# B&R Automation Studio project 2x1HWDemo (part 2)

### GlobalTypes.typ
```iecst
(*Main System Interface Types*)

TYPE
	MainIfTyp : 	STRUCT
		Cmd : MainIfCmdTyp;
		Par : MainIfParTyp;
		Cfg : MainIfCfgTyp;
		Status : MainIfStatusTyp;
	END_STRUCT;
	MainIfCmdTyp : 	STRUCT
		Power : BOOL;
		Start : BOOL;
		Stop : BOOL;
		Reset : BOOL;
	END_STRUCT;
	MainIfParTyp : 	STRUCT
		Tmp : USINT;
	END_STRUCT;
	MainIfCfgTyp : 	STRUCT
		ShuttleCount : USINT;
	END_STRUCT;
	MainIfStatusTyp : 	STRUCT
		PowerOn : BOOL;
		Running : BOOL;
		Error : BOOL;
	END_STRUCT;
END_TYPE

(*Process Info Interface*)

TYPE
	ProcessInfoIfTyp : 	STRUCT
		Cmd : ProcessInfoIfCmdTyp;
		Par : ProcessInfoIfParTyp;
		Sts : ProcessInfoIfStsTyp;
	END_STRUCT;
	ProcessInfoIfCmdTyp : 	STRUCT
		Enable : BOOL;
		ResetData : BOOL;
	END_STRUCT;
	ProcessInfoIfParTyp : 	STRUCT
		CurrentProductCount : UDINT;
	END_STRUCT;
	ProcessInfoIfStsTyp : 	STRUCT
		Enabled : BOOL;
		CurrentPPM : REAL;
		CurrentPPH : REAL;
		CurrentBlistersPerMinute : REAL;
		CurrentLayersPerMinute : REAL;
	END_STRUCT;
END_TYPE

(*6D Controller Interface Types*)

TYPE
	Acp6DCmdType : 	STRUCT
		Power : BOOL;
		ErrorReset : BOOL;
		GetErrorInfo : BOOL;
	END_STRUCT;
	Acp6DCtrlType : 	STRUCT
		Cmd : Acp6DCmdType;
		Status : Acp6DStatusType;
		Par : Acp6DParType;
	END_STRUCT;
	Acp6DParType : 	STRUCT
		Mode : McAcp6DMoveModeEnum;
		PathType : McAcp6DInPlaneMovePathEnum;
		Acceleration : REAL;
		EndVelocity : REAL;
		Velocity : REAL;
		ShuttleID : USINT;
		SegmentID : USINT;
		PositionX : REAL;
		PositionY : REAL;
	END_STRUCT;
	Acp6DStatusType : 	STRUCT
		Error : BOOL;
		ErrorID : DINT;
		Ready : BOOL;
		PowerOn : BOOL;
		ReadyToPowerOn : BOOL;
		ErrorCodes : ARRAY[0..8]OF DINT;
	END_STRUCT;
	Acp6DShuttleInfoType : 	STRUCT
		State : Acp6DShuttleStateInfoTyp;
		Force : Acp6DShuttleForceInfoTyp;
		Position : Acp6DShuttlePosInfoTyp;
	END_STRUCT;
	Acp6DShuttleStateInfoTyp : 	STRUCT
		Valid : BOOL;
		Value : McAcp6DShuttleStateEnum;
	END_STRUCT;
	Acp6DShuttlePosInfoTyp : 	STRUCT
		Valid : BOOL;
		Value : McAcp6DShPositionInfoType;
	END_STRUCT;
	Acp6DShuttleForceInfoTyp : 	STRUCT
		Valid : BOOL;
		Value : McAcp6DShForceInfoType;
	END_STRUCT;
END_TYPE

(*Shuttle Interface Types*)

TYPE
	gShuttleIfCmdTyp : 	STRUCT  (*Commands for controlling a shuttle*)
		Enable : BOOL; (*Command for enabling the control of a shuttle in the process*)
		Recover : BOOL; (*Command for a shuttle to start recovery*)
		NextStep : BOOL; (*Command for a shuttle to start the next step in the process*)
		ResetProductInfo : BOOL; (*Command to reset all the product info on a shuttle*)
		Stop : BOOL; (*Command to stop the process for a shuttle*)
	END_STRUCT;
	gShuttleIfCfgMacrosTyp : 	STRUCT  (*Structure of the macro IDs used for operation*)
		RobotProcessMacro : gShuttleIfMacroEnum; (*Macro ID used for sending a shuttle from the load station to the print station*)
	END_STRUCT;
	gShuttleIfParTyp : 	STRUCT  (*Parameters for the shuttle's operation*)
		NumLayers : USINT; (*Number of layers for this defined recipe*)
		MacroIDs : gShuttleIfCfgMacrosTyp; (*Macro's used for routing shuttles*)
	END_STRUCT;
	gShuttleIfConfigTyp : 	STRUCT  (*Configuration values for a shuttle*)
		ShuttleId : USINT; (*ShuttleID of this shuttle*)
	END_STRUCT;
	gShuttleIfMacroEnum :
		( (*Macro IDs that are used to denote which macro means what*)
		MACRO_ROBOT_PROCESS := 128, (*Macro ID used for sending a shuttle from the load station to the print station*)
		MACRO_RECOVERY_GROUP0 (*Macro ID used for recovering the group 0 shuttles*)
		);
	gShuttleIfDestEnum :
		( (*Destinations for a shuttle to move to*)
		DEST_LOAD, (*Destination Load station*)
		DEST_PRINT, (*Destination Printing station*)
		DEST_DOSE1, (*Destination Dose 1 station*)
		DEST_DOSE2, (*Destination Dose 2 station*)
		DEST_TAMP, (*Destination Tamping station*)
		DEST_UNLOAD (*Destination unload*)
		);
	ShStateEnum :
		(
		SH_OFF, (*Shuttle is in the off/idle state*)
		SH_INIT, (*Shuttle is in the initilization state*)
		SH_STARTUP, (*Shuttle is in the startup state*)
		SH_IDLE, (*Shuttle is in the idle state after having been recovered*)
		SH_MOVE_TO_ROBOT,
		SH_ROBOT,
		SH_OFFLOAD, (*Shuttle is currently being offloaded*)
		SH_ERROR := 65535 (*Shuttle is in the error state*)
		);
	gShuttleIfStatusTyp : 	STRUCT  (*Status information for the shuttle*)
		CurrentDestination : gShuttleIfDestEnum; (*Destination the shuttle is currently moving towards*)
		ShuttleInfo : Acp6DShuttleInfoType; (*CurrentStatus Information about the shuttle*)
		Error : BOOL; (*Shuttle is currently in an error state*)
		ErrorState : ShStateEnum; (*State the shuttle errored at*)
		Recovered : BOOL; (*Shuttle has been recovered*)
		CyclicPositionX : REAL;
	END_STRUCT;
	gShuttleIfTyp : 	STRUCT  (*Interface for controlling a shuttle*)
		Cmd : gShuttleIfCmdTyp; (*Commands to issue to a shuttle*)
		Par : gShuttleIfParTyp; (*Parameters for the process for this shuttle*)
		Cfg : gShuttleIfConfigTyp; (*Configuration values for this shuttle*)
		Status : gShuttleIfStatusTyp; (*Status information related to this shuttle*)
	END_STRUCT;
END_TYPE

(*Robot Interface Types*)

TYPE
	RobotIfTyp : 	STRUCT
		Cmds : RobotIfCmdsTyp;
		Pars : RobotIfParsTyp;
		Status : RobotIfStatusTyp;
	END_STRUCT;
	RobotIfCmdsTyp : 	STRUCT
		Admin : RobotIfAdminCmdsTyp;
		Process : RobotIfProcessCmdsTyp;
	END_STRUCT;
	RobotIfAdminCmdsTyp : 	STRUCT
		Power : BOOL;
		Home : BOOL;
		Reset : BOOL;
	END_STRUCT;
	RobotIfProcessCmdsTyp : 	STRUCT
		MoveToSync : BOOL;
		Sync : BOOL;
		UnSync : BOOL;
		Run : BOOL;
	END_STRUCT;
	RobotIfParsTyp : 	STRUCT
		SyncPosition : McPosType;
		SyncFrame : STRING[80];
		SyncFrameIdent : UDINT;
		MoveToSyncVel : LREAL;
		MoveToSyncAccel : LREAL;
		MoveToSyncDecel : LREAL;
		ShuttleIdx : USINT;
	END_STRUCT;
	RobotIfStatusTyp : 	STRUCT
		Synced : BOOL;
		Homed : BOOL;
		Powered : BOOL;
		AtSync : BOOL;
	END_STRUCT;
	SceneViewerTyp : 	STRUCT
		Cmds : SceneViewerCmdsTyp;
		Pars : SceneViewerParsTyp;
	END_STRUCT;
	SceneViewerCmdsTyp : 	STRUCT
		Record : BOOL;
		Clear : BOOL;
	END_STRUCT;
	SceneViewerParsTyp : 	STRUCT
		LineColor : SceneViewerColorTyp;
	END_STRUCT;
	SceneViewerColorTyp : 	STRUCT
		Red : REAL;
		Green : REAL;
		Blue : REAL;
	END_STRUCT;
END_TYPE

(*Sync Interface Types*)

TYPE
	SyncSecIfTyp : 	STRUCT
		Cmds : SyncSecCmdsIfTyp;
		Pars : USINT;
		Status : SyncSecIfStatusTyp;
	END_STRUCT;
	SyncSecCmdsIfTyp : 	STRUCT
		Admin : SyncSecIfAdminCmdsTyp;
		Proc : SyncSecIfProcCmdsTyp;
	END_STRUCT;
	SyncSecIfAdminCmdsTyp : 	STRUCT
		New_Member : USINT;
	END_STRUCT;
	SyncSecIfProcCmdsTyp : 	STRUCT
		Start : BOOL;
		Stop : BOOL;
		ReleaseSync : BOOL;
		ReleaseUnSync : BOOL;
	END_STRUCT;
	SyncSecIfStatusTyp : 	STRUCT
		Running : BOOL;
		SyncReady : BOOL;
		UnsyncReady : BOOL;
		Error : BOOL;
		AxisToSync : McAxisType;
	END_STRUCT;
	SyncSecStatusEnum :
		(
		SYNC_OFF,
		SYNC_INIT,
		SYNC_RUNNING,
		SYNC_STOPPING,
		SYNC_ERROR
		);
END_TYPE

(*Recovery Interface Type*)

TYPE
	Acp6DRecoveryIfTyp : 	STRUCT
		Cmd : Acp6DRecoveryCmdTyp;
		Par : Acp6DRecoveryParTyp;
		Sts : Acp6DRecoveryStsTyp;
	END_STRUCT;
	Acp6DRecoveryCmdTyp : 	STRUCT
		Recover : BOOL;
		Reset : BOOL;
	END_STRUCT;
	Acp6DRecoveryParTyp : 	STRUCT
		AutoDrivePositions : ARRAY[0..MAX_SHUTTLE_COUNT_ARRAY]OF Acp6DAutoDrivePosTyp;
		Vel : REAL;
		Accel : REAL;
	END_STRUCT;
	Acp6DRecoveryStsTyp : 	STRUCT
		Recovering : BOOL;
		ReadyToStartProc : BOOL;
		Done : BOOL;
		ShuttlesRecovered : BOOL;
		Error : BOOL;
	END_STRUCT;
	Acp6DAutoDrivePosTyp : 	STRUCT
		ShIdx : USINT;
		GroupNum : USINT; (*Group ID used for recovery. Lower group, lower priority*)
		X : REAL;
		Y : REAL;
	END_STRUCT;
END_TYPE

(***********************Station Types*)
(*Load Station Types*)

TYPE
	LoadStationIfTyp : 	STRUCT
		Cmd : LoadStationCmdTyp; (*Commands to the station*)
		Par : LoadStationParTyp; (*Paramters for the station's operation*)
		Cfg : LoadStationCfgTyp; (*Configuration values for the station*)
		Status : LoadStationStatusTyp; (*Status of the station*)
	END_STRUCT;
	LoadStationCmdTyp : 	STRUCT
		Enable : BOOL; (*Enables the process station*)
		Process : BOOL; (*Start a process for the station with the defined shuttle index*)
		Reset : BOOL; (*Resets the process from an any state*)
	END_STRUCT;
	LoadStationParTyp : 	STRUCT
		ShuttleIdx : USINT; (*Index in the gShuttle array for the shuttle in question*)
		WaitTime : TIME; (*Amount of time to wait for the load process*)
	END_STRUCT;
	LoadStationCfgTyp : 	STRUCT
		StationPos : StationPositionTyp; (*Station's center world position*)
	END_STRUCT;
	LoadStationStatusTyp : 	STRUCT
		Enabled : BOOL; (*Signal denoting the station is enabled and in an operational state*)
		Processing : BOOL; (*Signal denoting the station is currently operating on a shuttle*)
		Done : BOOL; (*Signal denoting the current operation has completed*)
		ReadyForNewShuttle : BOOL; (*Signal denoting the station is ready for a new shuttle*)
		Error : BOOL; (*Signal denoting the station has an error present*)
	END_STRUCT;
	StationPositionTyp : 	STRUCT
		X : REAL; (*Station's Global X position*)
		Y : REAL; (*Station's Global Y position*)
	END_STRUCT;
END_TYPE

(*Pick Place Types*)

TYPE
	posTyp : 	STRUCT
		X : LREAL;
		Y : LREAL;
		Z : LREAL;
	END_STRUCT;
	RobotPickPlaceParsTyp : 	STRUCT
		PickTune : pickTuneTyp;
		PlaceTune : pickTuneTyp;
		ReadyPos : posTyp;
		ProductSpeed : robotSpeedTyp;
		EmptySpeed : robotSpeedTyp;
	END_STRUCT;
	pickTuneTyp : 	STRUCT
		ApproachHeight : LREAL;
		DepartHeight : LREAL;
		XTune : LREAL;
		YTune : LREAL;
		ZTune : LREAL;
		Radius : LREAL;
		DwellTime : REAL;
	END_STRUCT;
	robotSpeedTyp : 	STRUCT
		Vel : REAL;
		Accel : REAL;
		Decel : REAL;
	END_STRUCT;
	RobotPickPlaceStatusTyp : 	STRUCT
		ProductOK : BOOL;
		ProductPresent : BOOL;
		AtSync : BOOL;
	END_STRUCT;
	RobotPickPlaceCfgTyp : 	STRUCT
		PlaceLoc : posTyp;
		PickLoc : posTyp;
		SyncLoc : posTyp;
	END_STRUCT;
	RobotPickPlaceTyp : 	STRUCT
		Run : BOOL;
		Sync : BOOL;
		Config : RobotPickPlaceCfgTyp;
		Pars : RobotPickPlaceParsTyp;
		Status : RobotPickPlaceStatusTyp;
	END_STRUCT;
END_TYPE
```

### Package Logical/Source/ShuttleCtrl - Package that contains code for controlling individual shuttles

### Program Logical/Source/ShuttleCtrl/ShCtrl (IEC)

#### Types.typ
```iecst
TYPE
	ShFbsTyp : 	STRUCT
		ShRunMacroFb : MC_BR_MacroRun_Acp6D; (*Execute a macro on the current shuttle*)
		ReadCyclicPos : MC_BR_ReadCyclicChAxis_Acp6D;
	END_STRUCT;
END_TYPE
```

#### Variables.var
```iecst
VAR
	i : USINT; (*Loop index*)
	shState : ARRAY[0..MAX_SHUTTLE_COUNT_ARRAY] OF ShStateEnum;
	shFbs : ARRAY[0..MAX_SHUTTLE_COUNT_ARRAY] OF ShFbsTyp;
	pDebugIf : REFERENCE TO gShuttleIfTyp;
	pDebugFbs : REFERENCE TO ShFbsTyp;
	pDebugState : REFERENCE TO ShStateEnum;
	debugIdx : USINT;
END_VAR
```

#### Cyclic.st
```iecst
PROGRAM _CYCLIC
	FOR i:= 0 TO gMainIf.Cfg.ShuttleCount - 1 DO

		CASE shState[i] OF
			SH_OFF:  //******************************************************************************** Shuttle is in the off/idle state
				IF gShuttleIf[i].Cmd.Enable THEN
					shState[i] := SH_INIT;
				ELSE

				END_IF
			SH_INIT:  //******************************************************************************** Shuttle is in the initilization state
				//In this state we could make any checks on the current shuttle process perhaps in order to aide in recovery?
				shFbs[i].ReadCyclicPos.Controller := ADR(gMcAcp6DController);
				shFbs[i].ReadCyclicPos.ChannelID := i + 1;
				shFbs[i].ReadCyclicPos.AxisID := 1;
				shFbs[i].ReadCyclicPos.Enable := TRUE;

				shState[i] := SH_STARTUP;
			SH_STARTUP:  //******************************************************************************** Shuttle is in the startup state
				//In this state maybe we have triggered recovery and we're waiting for the autodrive to complete
				IF shFbs[i].ReadCyclicPos.Valid THEN
					shState[i] := SH_IDLE;
				END_IF
			SH_IDLE:  //******************************************************************************** Shuttle is in the idle state
				IF gShuttleIf[i].Cmd.NextStep THEN
					gShuttleIf[i].Cmd.NextStep := FALSE;
					//Evaluate the current step to determine what the next step should be
					shFbs[i].ShRunMacroFb.Controller := ADR(gMcAcp6DController);
					shFbs[i].ShRunMacroFb.ShuttleID := gShuttleIf[i].Cfg.ShuttleId;
					shFbs[i].ShRunMacroFb.MacroID := UDINT_TO_USINT(gShuttleIf[i].Par.MacroIDs.RobotProcessMacro);
					shFbs[i].ShRunMacroFb.Execute := TRUE;
					gShuttleIf[i].Status.CurrentDestination := DEST_LOAD;
					LogDebug(gAuditTrail,i,"Sent to Robot");

					shState[i] := SH_MOVE_TO_ROBOT;
				END_IF
			SH_MOVE_TO_ROBOT:  //******************************************************************************** Shuttle is moving to the load position
				IF shFbs[i].ShRunMacroFb.Error THEN
					gShuttleIf[i].Status.Error := TRUE;
					gShuttleIf[i].Status.ErrorState := shState[i];
					shState[i] := SH_ERROR;
				ELSIF shFbs[i].ShRunMacroFb.Acknowledge THEN //Check to see if the shuttle is ready to sync with the robot
					gLoadStationIf.Par.ShuttleIdx := i;
					gLoadStationIf.Cmd.Process := TRUE;

					LogDebug(gAuditTrail,i,"Arrived at Robot");

					shFbs[i].ShRunMacroFb.Execute := FALSE;
					shState[i] := SH_ROBOT;
				END_IF
			SH_ROBOT:  //******************************************************************************** Shuttle is currently being loaded
				//Station has control on the shuttle during this section
				IF gShuttleIf[i].Cmd.NextStep THEN
					gLoadStationIf.Cmd.Process := FALSE; //Respond to the Load station we're done

					gShuttleIf[i].Cmd.NextStep := FALSE;
					gShuttleIf[i].Status.CurrentDestination := DEST_PRINT;

					LogDebug(gAuditTrail,i,"Finished with Robot");

					shState[i] := SH_MOVE_TO_ROBOT;
				END_IF

			SH_ERROR: //******************************************************************************** Shuttle is in the error state

		END_CASE;
		shFbs[i].ShRunMacroFb();

		IF gShuttleIf[i].Cmd.ResetProductInfo THEN
			gShuttleIf[i].Status.Error := FALSE;
			gShuttleIf[i].Status.ErrorState := 0;
			gShuttleIf[i].Cmd.ResetProductInfo := FALSE;
		END_IF
	END_FOR;
	pDebugIf ACCESS ADR(gShuttleIf[debugIdx]);
	pDebugState ACCESS ADR(shState[debugIdx]);
	pDebugFbs ACCESS ADR(shFbs[debugIdx]);

END_PROGRAM
```

#### Init.st
```iecst
PROGRAM _INIT
	FOR i:=0 TO MAX_SHUTTLE_COUNT-1 DO
		gShuttleIf[i].Par.MacroIDs.RobotProcessMacro := MACRO_ROBOT_PROCESS;

	END_FOR;
END_PROGRAM
```

### Program Logical/Source/ShuttleCtrl/Recovery (IEC)

#### Init.st
```iecst
PROGRAM _INIT
	g6DRecoveryIf.Par.Vel := 1;
	g6DRecoveryIf.Par.Accel := 10;

	//************************************************************************* Shuttle 1
	g6DRecoveryIf.Par.AutoDrivePositions[0].ShIdx := 0;
	g6DRecoveryIf.Par.AutoDrivePositions[0].GroupNum := 0;
	g6DRecoveryIf.Par.AutoDrivePositions[0].X := 0.12;
	g6DRecoveryIf.Par.AutoDrivePositions[0].Y := 0.12;
	//************************************************************************* Shuttle 2
	g6DRecoveryIf.Par.AutoDrivePositions[1].ShIdx := 1;
	g6DRecoveryIf.Par.AutoDrivePositions[1].GroupNum := 0;
	g6DRecoveryIf.Par.AutoDrivePositions[1].X := 0.36;
	g6DRecoveryIf.Par.AutoDrivePositions[1].Y := 0.12;

END_PROGRAM
```

### Program Logical/Source/ShuttleCtrl/KalmanTesting (IEC)

#### Types.typ
```iecst
TYPE
	WeighTyp : 	STRUCT
		TareWeight : REAL;
		ExpectedWeight : REAL;
		Error : REAL;
		CalculatedExpectedForce : REAL;
		CalcWeight : REAL;
		TriggerThreshold : REAL;
	END_STRUCT;
END_TYPE
```

#### Variables.var
```iecst
VAR
	readCyclicForceFb : MC_BR_ReadCyclicChAxis_Acp6D;
	weighKalman : WFPredictiveFilter;
	WeighFb : MC_BR_GetPayload_Acp6D;
	OutputCovertedToWeight : ARRAY[0..1] OF LREAL;
	filterTest : BOOL;
	WeightTest : BOOL;
	enableFilters : BOOL;
	state : INT;
	KalmanFb : ARRAY[0..1] OF MTFilterKalman;
	ExpectedWeight : REAL;
	finalWeighKalmanFb : WFPredictiveFilter;
	Reset : BOOL;
	rawWeight : REAL;
	shiftedWeight : REAL;
	weightValues : WeighTyp;
END_VAR
```

#### Cyclic.st
```iecst
PROGRAM _CYCLIC
	//rawWeight := gShuttleIf[0].Status.ShuttleInfo.Force.Value.Fz / 9.81 * 1000.0;
	rawWeight := readCyclicForceFb.Value / 9.81 * 1000.0;
	weightValues.CalcWeight := rawWeight * 1.1588+70.798-weightValues.TareWeight;
	CASE state OF
		0:
			IF enableFilters THEN

				KalmanFb[1].Enable := TRUE;
				weighKalman.Enable := TRUE;

				readCyclicForceFb.Enable := TRUE;
				readCyclicForceFb.ChannelID := 2;
				readCyclicForceFb.AxisID := 3;
				readCyclicForceFb.Controller := ADR(gMcAcp6DController);
				state := 5;
			END_IF
		5:
			IF readCyclicForceFb.Valid THEN
				state := 10;
			END_IF
		10:
			KalmanFb[1].SystemOutput := rawWeight;

			weighKalman.Input := weightValues.CalcWeight;

			IF weighKalman.Output > weightValues.ExpectedWeight * weightValues.TriggerThreshold THEN
				finalWeighKalmanFb.Enable := TRUE;
				finalWeighKalmanFb.Input := weightValues.ExpectedWeight;
				KalmanFb[0].Enable := TRUE;
				KalmanFb[0].SystemOutput := weightValues.ExpectedWeight;
				state := 11;
			END_IF

			IF NOT enableFilters THEN
				KalmanFb[0].Enable := FALSE;
				KalmanFb[1].Enable := FALSE;
				weighKalman.Enable := FALSE;

				state := 0;
			END_IF
		11:
			weighKalman.Input := weightValues.CalcWeight;
			finalWeighKalmanFb.Input := weighKalman.Output;
			KalmanFb[0].SystemOutput := weightValues.CalcWeight;
			IF Reset OR weighKalman.Output < weightValues.ExpectedWeight * weightValues.TriggerThreshold THEN
				Reset := FALSE;
				finalWeighKalmanFb.Enable := FALSE;
				state := 10;
			END_IF
		20:
		//Sigma A should be standard deviation of the process, so if the pill weighing process, what is the deviation for missed pills?

		//Use single kalman w/ correct Z (Z is the standard deviation is  from your raw signal)
		//	A  is very high so that the signal follows raw relatively closely (lots of process noise)
		//When value reaches window of expected known
		//Start 2nd kalman w/ same Z and much lower A to remove the process noise
			//AND set the initial value for the expected weight to help converge faster
	END_CASE;

	KalmanFb[0]();
	KalmanFb[1]();
	readCyclicForceFb();
	weighKalman();
	finalWeighKalmanFb();

	OutputCovertedToWeight[0] := KalmanFb[0].FilteredOutput[0];
	OutputCovertedToWeight[1] := KalmanFb[1].FilteredOutput[0];

	IF WeightTest THEN
		WeighFb.Controller := ADR(gMcAcp6DController);
		WeighFb.ShuttleID := 1;
		WeighFb.Execute := NOT WeighFb.Valid;
	END_IF
	WeighFb();
END_PROGRAM
```

#### Init.st
```iecst
PROGRAM _INIT
	KalmanFb[0].Numerator[0] := 1;
	KalmanFb[0].Denominator[1] := 1;
	KalmanFb[0].NoiseReduction := 3;
	KalmanFb[1].Numerator[0] := 1;
	KalmanFb[1].Denominator[1] := 1;
	KalmanFb[1].NoiseReduction := 3;

	weighKalman.Time := 0.005;
	weighKalman.SigmaA := 10000.0;
	weighKalman.SigmaZ := 4.4;
	weighKalman.Alpha := 1.0;

	finalWeighKalmanFb.Time := 0.005;
	finalWeighKalmanFb.SigmaA := 1.0;
	finalWeighKalmanFb.SigmaZ := 4.4;
	finalWeighKalmanFb.Alpha := 1.01;
	weightValues.TareWeight := 695.0;
	weightValues.ExpectedWeight := 500;
	weightValues.TriggerThreshold := 0.95;
	weightValues.CalculatedExpectedForce := weightValues.TareWeight + weightValues.ExpectedWeight + weightValues.Error;
END_PROGRAM
```

### Program Logical/Source/ProcessStations/LoadStation (IEC)

#### Types.typ
```iecst
TYPE
	LoadStationStateEnum :
		(
		LOAD_OFF, (*Load station is currently disabled*)
		LOAD_INIT, (*Load station is initalizing*)
		LOAD_HOME_MASTER, (*Load station need to home the master axis*)
		LOAD_WAIT_FOR_SHUTTLE, (*Load station is waiting for a shuttle to be present*)
		LOAD_LOADING, (*Load station is loading product onto a shuttle*)
		LOAD_DONE, (*Load station is done with the load process*)
		LOAD_ERROR (*Load station had an error*)
		);
	LoadStationFbTyp : 	STRUCT
		LoadTimerFb : TON;
	END_STRUCT;
END_TYPE
```

#### Cyclic.st
```iecst
PROGRAM _CYCLIC
	CASE state OF
		LOAD_OFF: //********************************************************************************Load station is currently disabled
			IF gLoadStationIf.Cmd.Enable THEN
				state := LOAD_INIT;
			END_IF
		LOAD_INIT: //********************************************************************************Load station is initalizing

				gLoadStationIf.Status.ReadyForNewShuttle := TRUE;
				gLoadStationIf.Status.Enabled := TRUE;
				state := LOAD_WAIT_FOR_SHUTTLE;

		LOAD_WAIT_FOR_SHUTTLE: //********************************************************************************Load station is waiting for a shuttle to be present
			IF NOT gLoadStationIf.Cmd.Enable THEN
				gLoadStationIf.Status.ReadyForNewShuttle := FALSE;
				gLoadStationIf.Status.Enabled := FALSE;
				state := LOAD_OFF;
			ELSIF gLoadStationIf.Par.ShuttleIdx <> STATION_IS_EMPTY AND gLoadStationIf.Cmd.Process THEN
				gLoadStationIf.Status.ReadyForNewShuttle := FALSE;
				gLoadStationIf.Status.Processing := TRUE;

				LoadStationFbs.LoadTimerFb.IN := TRUE;
				LoadStationFbs.LoadTimerFb.PT := gLoadStationIf.Par.WaitTime;

				state := LOAD_LOADING;
			END_IF
		LOAD_LOADING: //********************************************************************************Load station is loading product onto a shuttle
			IF LoadStationFbs.LoadTimerFb.Q THEN
				LoadStationFbs.LoadTimerFb.IN := FALSE;

				gLoadStationIf.Status.Processing := FALSE;
				gShuttleIf[gLoadStationIf.Par.ShuttleIdx].Cmd.NextStep := TRUE;
				gLoadStationIf.Status.Done := TRUE;

				state := LOAD_DONE;
			END_IF
		LOAD_DONE: //********************************************************************************Load station is done with the load process
			IF NOT gLoadStationIf.Cmd.Enable THEN
				gLoadStationIf.Status.Done := FALSE;
				gLoadStationIf.Status.Enabled := FALSE;
				gLoadStationIf.Status.ReadyForNewShuttle := FALSE;
				state := LOAD_OFF;
			ELSIF NOT gLoadStationIf.Cmd.Process THEN
				gLoadStationIf.Par.ShuttleIdx := STATION_IS_EMPTY;
				gLoadStationIf.Status.Done := FALSE;
				gLoadStationIf.Status.ReadyForNewShuttle := FALSE;
				gLoadStationIf.Status.ReadyForNewShuttle := TRUE;

				state := LOAD_WAIT_FOR_SHUTTLE;
			END_IF

		LOAD_ERROR: //********************************************************************************Load station had an error
			IF gLoadStationIf.Cmd.Reset THEN
				gLoadStationIf.Cmd.Reset := FALSE;

				gLoadStationIf.Status.Done := FALSE;
				gLoadStationIf.Status.Enabled := FALSE;
				gLoadStationIf.Status.Error := FALSE;
				gLoadStationIf.Status.Processing := FALSE;
				gLoadStationIf.Status.ReadyForNewShuttle := FALSE;

				gLoadStationIf.Par.ShuttleIdx := STATION_IS_EMPTY;
				IF gLoadStationIf.Cmd.Enable THEN
					state := LOAD_INIT;
				ELSE
					state := LOAD_OFF;
				END_IF
			END_IF
	END_CASE;

	 LoadStationFbs.LoadTimerFb();
END_PROGRAM
```

### Program Logical/Source/ProcessStations/DoseStation

#### Cyclic.st
```iecst
PROGRAM _CYCLIC
	CASE state OF
		DOSE_OFF: //********************************************************************************Dose station is currently disabled
			IF pDoseIf.Cmd.Enable THEN
				state := DOSE_INIT;
			END_IF
		DOSE_INIT: //********************************************************************************Dose station is initalizing
			pDoseIf.Status.ReadyForNewShuttle := TRUE;
			pDoseIf.Status.Enabled := TRUE;
			state := DOSE_WAIT_FOR_SHUTTLE;
		DOSE_WAIT_FOR_SHUTTLE: //********************************************************************************Dose station is waiting for a shuttle to be present
			IF NOT pDoseIf.Cmd.Enable THEN
				pDoseIf.Status.ReadyForNewShuttle := FALSE;
				pDoseIf.Status.Enabled := FALSE;
				state := DOSE_OFF;
			ELSIF pDoseIf.Par.ShuttleIdx <> STATION_IS_EMPTY AND pDoseIf.Cmd.Process THEN
				pDoseIf.Status.ReadyForNewShuttle := FALSE;
				pDoseIf.Status.Processing := TRUE;

				DoseStationFbs.DoseMoveFb.Controller := ADR(gMcAcp6DController);
				DoseStationFbs.DoseMoveFb.ShuttleID := gShuttleIf[pDoseIf.Par.ShuttleIdx].Cfg.ShuttleId;
				DoseStationFbs.DoseMoveFb.Mode := mcACP6D_MOVE_RELATIVE;
				DoseStationFbs.DoseMoveFb.Path := mcACP6D_PATH_DIRECT;
				DoseStationFbs.DoseMoveFb.Velocity := pDoseIf.Par.Vel;
				DoseStationFbs.DoseMoveFb.EndVelocity := pDoseIf.Par.EndVel;
				DoseStationFbs.DoseMoveFb.Acceleration := pDoseIf.Par.Accel;
				DoseStationFbs.DoseMoveFb.PositionX := (pDoseIf.Par.FirstCavityPosition.DistX);
				DoseStationFbs.DoseMoveFb.PositionY := -(pDoseIf.Par.FirstCavityPosition.DistY); //Made negative as we're moving in negative Z
				DoseStationFbs.DoseMoveFb.Execute := TRUE;
//
//				msgType := "";
//				msgMsg := "";
//				tmp := STRING_TO_WSTRING(taskName);
//				brwcscat(ADR(msgType),ADR(tmp));
//				brwcscat(ADR(msgType),ADR(":FirstMove:Sh"));
//				tmp := USINT_TO_WSTRING(gShuttleIf[pDoseIf.Par.ShuttleIdx].Cfg.ShuttleId);
//				brwcscat(ADR(msgType),ADR(tmp));
//				tmp := "";
//				msgMsg := "X:";
//				tmp := REAL_TO_WSTRING(DoseStationFbs.DoseMoveFb.PositionX);
//				brwcscat(ADR(msgMsg),ADR(tmp));
//				brwcscat(ADR(msgMsg),ADR(" Y:"));
//				tmp := REAL_TO_WSTRING(DoseStationFbs.DoseMoveFb.PositionY);
//				brwcscat(ADR(msgMsg),ADR(tmp));
//				MpAuditCustomEvent(gAuditTrail,"DEBUG",msgType,msgMsg);

				state := DOSE_INDEX_SHUTTLE;
			END_IF
		DOSE_INDEX_SHUTTLE: //******************************************************************************** Dose station is indexing to the next dosing position
			IF DoseStationFbs.DoseMoveFb.Error THEN
				pDoseIf.Status.Error := TRUE;

				state := DOSE_ERROR;
			ELSIF DoseStationFbs.DoseMoveFb.Done THEN
				DoseStationFbs.DoseMoveFb.Execute:= FALSE;

				DoseStationFbs.WaitTimer.IN := TRUE;
				DoseStationFbs.WaitTimer.PT := pDoseIf.Par.WaitTime;

				state := DOSE_DOSING;
			END_IF
		DOSE_DOSING: //********************************************************************************Dose station is preforming the dosing process
			IF DoseStationFbs.WaitTimer.Q THEN
				DoseStationFbs.WaitTimer.IN := FALSE;

				currentRow := currentRow + 1;
				IF currentRow > pDoseIf.Par.NumRowsOfCavities THEN
					gShuttleIf[pDoseIf.Par.ShuttleIdx].Cmd.NextStep := TRUE;
					pDoseIf.Status.Done := TRUE;
					pDoseIf.Status.Processing := FALSE;

					state := DOSE_DONE;
				ELSE
					DoseStationFbs.DoseMoveFb.Controller := ADR(gMcAcp6DController);
					DoseStationFbs.DoseMoveFb.ShuttleID := gShuttleIf[pDoseIf.Par.ShuttleIdx].Cfg.ShuttleId;
					DoseStationFbs.DoseMoveFb.Mode := mcACP6D_MOVE_RELATIVE;
					DoseStationFbs.DoseMoveFb.Path := mcACP6D_PATH_DIRECT;
					DoseStationFbs.DoseMoveFb.Velocity := pDoseIf.Par.Vel;
					DoseStationFbs.DoseMoveFb.EndVelocity := pDoseIf.Par.EndVel;
					DoseStationFbs.DoseMoveFb.Acceleration := pDoseIf.Par.Accel;
					DoseStationFbs.DoseMoveFb.PositionX := (pDoseIf.Par.SpaceBetweenCavities.DistX);
					DoseStationFbs.DoseMoveFb.PositionY := -(pDoseIf.Par.SpaceBetweenCavities.DistY); //Made negative as we're moving in negative Z
					DoseStationFbs.DoseMoveFb.Execute := TRUE;

					state := DOSE_INDEX_SHUTTLE;
				END_IF
			END_IF
		DOSE_DONE: //********************************************************************************Dose station is done with the load process
			IF NOT pDoseIf.Cmd.Enable THEN
				pDoseIf.Status.Enabled := FALSE;
				pDoseIf.Status.ReadyForNewShuttle := FALSE;
				currentRow := 0;

				state := DOSE_OFF;
			ELSIF NOT pDoseIf.Cmd.Process THEN
				pDoseIf.Status.Done := FALSE;
				currentRow := 0;

				pDoseIf.Par.ShuttleIdx := STATION_IS_EMPTY;
				pDoseIf.Status.ReadyForNewShuttle := FALSE;
				pDoseIf.Status.ReadyForNewShuttle := TRUE;

				state := DOSE_WAIT_FOR_SHUTTLE;
			END_IF
		DOSE_ERROR: //********************************************************************************Dose station had an error
			IF pDoseIf.Cmd.Reset THEN
				pDoseIf.Cmd.Reset := FALSE;

				pDoseIf.Par.ShuttleIdx := STATION_IS_EMPTY;

				currentRow := 0;

				pDoseIf.Status.Done := FALSE;
				pDoseIf.Status.Error := FALSE;
				pDoseIf.Status.Processing := FALSE;
				pDoseIf.Status.ReadyForNewShuttle := FALSE;
				pDoseIf.Status.Enabled := FALSE;

				DoseStationFbs.DoseMoveFb.Execute := FALSE;
				DoseStationFbs.WaitTimer.IN := FALSE;

				IF pDoseIf.Cmd.Enable THEN
					state := DOSE_INIT;
				ELSE
					state := DOSE_OFF;
				END_IF
			END_IF
	END_CASE;

	DoseStationFbs.DoseMoveFb();
	DoseStationFbs.WaitTimer();
END_PROGRAM
```

### Package Logical/Source/Main - Package that contains the main entry point to the machine

### Program Logical/Source/Main/Main

#### Types.typ
```iecst
TYPE
	MainStatesEnum :
		(
		MAIN_OFF,
		MAIN_INIT,
		MAIN_RECOVERING,
		MAIN_READY,
		MAIN_STARTING_ROBOT,
		MAIN_STARTING,
		MAIN_RUNNING,
		MAIN_STOPPING,
		MAIN_ERROR
		);
END_TYPE
```

#### Cyclic.st
```iecst
PROGRAM _CYCLIC
	IF gAcp6DCtrlIf.Status.Error THEN
		state := MAIN_ERROR;
	END_IF

	CASE state OF
		MAIN_OFF: //******************************************************************************** Main Off State
			IF gMainIf.Cmd.Power THEN
				gAcp6DCtrlIf.Cmd.Power := TRUE;

				state := MAIN_INIT;
			END_IF
		MAIN_INIT: //******************************************************************************** Main Initializing State
			IF gAcp6DCtrlIf.Status.PowerOn AND gAcp6DCtrlIf.Status.Ready THEN
				gMainIf.Status.PowerOn := TRUE;
				g6DRecoveryIf.Cmd.Recover := TRUE;

				state := MAIN_RECOVERING;
			ELSIF NOT gMainIf.Cmd.Power THEN
				gAcp6DCtrlIf.Cmd.Power := FALSE;
				state := MAIN_OFF;
			END_IF
		MAIN_RECOVERING: //******************************************************************************** Main Recovery State
			IF g6DRecoveryIf.Sts.ReadyToStartProc THEN
				g6DRecoveryIf.Cmd.Recover := FALSE;

				state := MAIN_READY;
			END_IF
		MAIN_READY://******************************************************************************** Main Ready State
			IF gMainIf.Cmd.Start THEN
				gProcessInfoIf.Cmd.Enable := TRUE;
				CmdShEnable(TRUE, ADR(gShuttleIf), gMainIf.Cfg.ShuttleCount);

				gRobotIf.Cmds.Admin.Power := TRUE;

				state := MAIN_STARTING;
			ELSIF NOT gMainIf.Cmd.Power THEN
				gMainIf.Status.PowerOn := FALSE;
				gAcp6DCtrlIf.Cmd.Power := FALSE;
				state := MAIN_OFF;
			END_IF
		MAIN_STARTING://******************************************************************************** Main Starting State

			gMainIf.Cmd.Start := FALSE;
			state := MAIN_RUNNING;

		MAIN_RUNNING: //******************************************************************************** Main Running State
			IF gMainIf.Cmd.Stop THEN

				state := MAIN_STOPPING;
			END_IF
		MAIN_STOPPING: //******************************************************************************** Main Stopping State

			gMainIf.Cmd.Stop := FALSE;

			FOR i:=0 TO gMainIf.Cfg.ShuttleCount - 1 DO
				gShuttleIf[i].Status.Recovered := FALSE;
			END_FOR;

			state := MAIN_READY;

		MAIN_ERROR: //******************************************************************************** Main Error State
			IF gMainIf.Cmd.Reset THEN
				gMainIf.Cmd.Reset := FALSE;
				gAcp6DCtrlIf.Cmd.ErrorReset := TRUE;

				state := MAIN_OFF;
			END_IF
	END_CASE;

END_PROGRAM
```

#### Init.st
```iecst
PROGRAM _INIT
	gMainIf.Cfg.ShuttleCount := 2;

	//Used to initialize the shuttle indecies.
	FOR i:=0 TO gMainIf.Cfg.ShuttleCount-1 DO
		gShuttleIf[i].Cfg.ShuttleId := i + 1;
	END_FOR;

END_PROGRAM
```

### Package Logical/Source/6DCtrl - Package containing the main logic for controlling the 6D system as a whole

### Program Logical/Source/6DCtrl/6DCtrl

#### Types.typ
```iecst
TYPE
	Acp6DStateEnum :
		( (*6D Control States*)
		ACP6D_RESET, (*Reset the 6D controller state*)
		ACP6D_POWER_OFF, (*System Power Off state*)
		ACP6D_INACTIVE, (*System inactive state*)
		ACP6D_POWER_ON, (*Powering on the system state*)
		ACP6D_WAIT_ACTIVATION, (*waiting for activation (needed for autoID)*)
		ACP6D_INIT_MACRO, (*Waiting for the initalization of the macros to be done*)
		ACP6D_CFG_CYCLIC_CHANNEL, (*Configure the cyclic channel*)
		ACP6D_READY, (*System Ready for operation*)
		ACP6D_ERROR := 255 (*System in an error state*)
		);
	Sys6DCtrlFbTyp : 	STRUCT
		AutoRefreshFB : MC_BR_AutoRefresh_Acp6D; (*FB that auto refreshes the 6D data*)
		PowerOnFb : MC_BR_SysPowerOn_Acp6D; (*FB to power on the 6D controller/system*)
		PowerOffFb : MC_BR_SysPowerOff_Acp6D; (*FB to power off the 6D controller/system*)
		SysReadStateFb : MC_BR_SysReadState_Acp6D; (*FB to read the state of the 6D controller*)
		ShReadPositionFb : ARRAY[0..MAX_SHUTTLE_COUNT_ARRAY]OF MC_BR_ShReadPosition_Acp6D; (*FB(s) to read the position of the shuttles*)
		ShReadForceFb : ARRAY[0..MAX_SHUTTLE_COUNT_ARRAY]OF MC_BR_ShReadForce_Acp6D; (*FB(s) to read the force acting on the shuttle*)
		ShReadState : ARRAY[0..MAX_SHUTTLE_COUNT_ARRAY]OF MC_BR_ShReadState_Acp6D; (*FB(s) to read the states of the shuttles*)
		GetErrorCodesFb : MC_BR_GetErrorCode_Acp6D; (*FB to read the error codes on the 6D controller*)
		CfgReadCyclicPos : MC_BR_ConfigReadCyclicCh_Acp6D; (*FB to configure the reading of the cyclic channels for the system*)
	END_STRUCT;
END_TYPE
```

#### Variables.var
```iecst
VAR
	Fbs : Sys6DCtrlFbTyp; (*Function Blocks to Ctrl 6D system*)
	state : Acp6DStateEnum; (*Acp6d state*)
	i : USINT; (*Loop index counter*)
	filterTest : BOOL;
END_VAR
```

#### Cyclic.st
```iecst
PROGRAM _CYCLIC

	IF((Fbs.SysReadStateFb.Valid AND Fbs.SysReadStateFb.State = mcACP6D_STATE_ERROR) AND (state <> ACP6D_ERROR))THEN
		state := ACP6D_ERROR;
	END_IF;

	CASE state OF
		ACP6D_RESET: 	//******************************************************************************** 6D Reset State
			IF(Fbs.SysReadStateFb.Valid AND (Fbs.SysReadStateFb.State = mcACP6D_STATE_INACTIVE))THEN
				state := ACP6D_INACTIVE;
			ELSIF(Fbs.SysReadStateFb.State = mcACP6D_STATE_OPERATION)THEN
				state := ACP6D_POWER_OFF;
			END_IF;

		ACP6D_POWER_OFF: 	//******************************************************************************** 6D Power off commanding State
			Fbs.PowerOffFb.Execute := TRUE;
			IF(Fbs.PowerOffFb.Acknowledge AND (Fbs.SysReadStateFb.Valid AND Fbs.SysReadStateFb.State = mcACP6D_STATE_INACTIVE))THEN
				gAcp6DCtrlIf.Status.PowerOn := FALSE;
				Fbs.PowerOffFb.Execute 	:= FALSE;
				state := ACP6D_INACTIVE;
			ELSIF(Fbs.PowerOffFb.Error)THEN
				Fbs.PowerOffFb.Execute 	:= FALSE;
				gAcp6DCtrlIf.Status.ErrorID := Fbs.PowerOffFb.ErrorID;
				state := ACP6D_ERROR;
			END_IF;

		ACP6D_INACTIVE:	 	//******************************************************************************** 6D Inactive/Power Off state
			IF(gAcp6DCtrlIf.Cmd.Power)THEN
				Fbs.PowerOnFb.Execute := TRUE;
				//MpAuditCustomEvent(gAuditTrail,"INFO","Acp6DSys","Power On Command Issued");
				state := ACP6D_POWER_ON;
			END_IF;

		ACP6D_POWER_ON: 	//******************************************************************************** 6D Power on Commanding State
			IF Fbs.PowerOnFb.Error THEN
				gAcp6DCtrlIf.Status.ErrorID := Fbs.PowerOnFb.ErrorID;
				state := ACP6D_ERROR;
			ELSIF(Fbs.PowerOnFb.Acknowledge AND (Fbs.SysReadStateFb.Valid AND (Fbs.SysReadStateFb.State > mcACP6D_STATE_INACTIVE)))THEN
				//MpAuditCustomEvent(gAuditTrail,"INFO","Acp6DSys","Powered On");
				Fbs.PowerOnFb.Execute := FALSE;
				state := ACP6D_WAIT_ACTIVATION;
			END_IF;

			//Necessary state when using Absolute ID.
		ACP6D_WAIT_ACTIVATION: 	//******************************************************************************** 6D Waiting for Activation of Shuttles State
			IF(Fbs.SysReadStateFb.Valid)THEN
				IF(Fbs.SysReadStateFb.State = mcACP6D_STATE_OPERATION)THEN
					gAcp6DCtrlIf.Status.PowerOn := TRUE;
					state := ACP6D_INIT_MACRO;
				ELSIF(Fbs.SysReadStateFb.State = mcACP6D_STATE_INACTIVE)THEN
					state := ACP6D_INACTIVE; // Error during Activating state; Can happen in Absolute ID mode.
					gAcp6DCtrlIf.Cmd.Power := FALSE;
				END_IF;
			END_IF;
		ACP6D_INIT_MACRO: 	//******************************************************************************** 6D Wait for Macro initilization State
			IF gMacroLoadIf.Status.AllMacrosLoaded THEN
				gMacroLoadIf.Cmd.LoadAll := FALSE;

				//This is hard coded for 2 axes to get the X position cyclically for the two FBs
				Fbs.CfgReadCyclicPos.Controller := ADR(gMcAcp6DController);
				Fbs.CfgReadCyclicPos.NumberOfChannels := 1;
				Fbs.CfgReadCyclicPos.ChannelID[0] := 1;
				Fbs.CfgReadCyclicPos.FeedbackMode[0] := mcACP6D_READ_CYCLIC_POSITION;
				Fbs.CfgReadCyclicPos.ShuttleID[0] := 1;
				Fbs.CfgReadCyclicPos.ShuttleID[1] := 2;
				Fbs.CfgReadCyclicPos.Execute := TRUE;

				state := ACP6D_CFG_CYCLIC_CHANNEL;
			ELSE
				gMacroLoadIf.Cmd.LoadAll := TRUE;
			END_IF
		ACP6D_CFG_CYCLIC_CHANNEL: 	//******************************************************************************** 6D Confiugring the cyclic channel reads
			IF Fbs.CfgReadCyclicPos.Error THEN
				gAcp6DCtrlIf.Status.Error := TRUE;
				gAcp6DCtrlIf.Status.ErrorID := Fbs.CfgReadCyclicPos.ErrorID;

				state := ACP6D_ERROR;
			ELSIF Fbs.CfgReadCyclicPos.Done THEN
				Fbs.CfgReadCyclicPos.Execute := FALSE;

				state := ACP6D_READY;
			END_IF
		ACP6D_READY: 	//******************************************************************************** 6D Ready/Running State
			IF(NOT gAcp6DCtrlIf.Cmd.Power)THEN
				gMacroLoadIf.Cmd.Reset := TRUE;
				state := ACP6D_POWER_OFF;
			END_IF;

		ACP6D_ERROR: 	//******************************************************************************** 6D Error State
			gAcp6DCtrlIf.Status.PowerOn := FALSE;
			IF(gAcp6DCtrlIf.Cmd.ErrorReset)THEN
				IF(Fbs.SysReadStateFb.State<>mcACP6D_STATE_ERROR)THEN
					gAcp6DCtrlIf.Cmd.ErrorReset := FALSE;
					state := ACP6D_RESET;
				ELSE
					Fbs.PowerOffFb.Execute := TRUE;	 // Reset error with power off.
					IF(Fbs.PowerOffFb.Acknowledge)THEN
						gMacroLoadIf.Cmd.Reset := TRUE;
						Fbs.PowerOffFb.Execute 	:= FALSE;
					ELSIF(Fbs.PowerOffFb.Error)THEN
						gAcp6DCtrlIf.Cmd.ErrorReset := FALSE;
						Fbs.PowerOffFb.Execute 	:= FALSE;
						gAcp6DCtrlIf.Status.ErrorID := Fbs.PowerOffFb.ErrorID;
						state := ACP6D_ERROR;
					END_IF;
				END_IF;
			END_IF;
	END_CASE;

	FOR i:=0 TO gMainIf.Cfg.ShuttleCount - 1 DO
		Fbs.ShReadPositionFb[i].Controller := ADR(gMcAcp6DController);
		Fbs.ShReadPositionFb[i].Enable := TRUE;
		Fbs.ShReadPositionFb[i].ShuttleID := gShuttleIf[i].Cfg.ShuttleId;
		Fbs.ShReadPositionFb[i]();

		Fbs.ShReadForceFb[i].Controller := ADR(gMcAcp6DController);
		Fbs.ShReadForceFb[i].Enable := TRUE;
		Fbs.ShReadForceFb[i].ShuttleID := gShuttleIf[i].Cfg.ShuttleId;
		Fbs.ShReadForceFb[i]();

		Fbs.ShReadState[i].Controller := ADR(gMcAcp6DController);
		Fbs.ShReadState[i].Enable := TRUE;
		Fbs.ShReadState[i].ShuttleID := gShuttleIf[i].Cfg.ShuttleId;
		Fbs.ShReadState[i]();

		gShuttleIf[i].Status.ShuttleInfo.Force.Value := Fbs.ShReadForceFb[i].ForceInfo;
		gShuttleIf[i].Status.ShuttleInfo.Force.Valid := Fbs.ShReadForceFb[i].Valid;
		gShuttleIf[i].Status.ShuttleInfo.Position.Value := Fbs.ShReadPositionFb[i].PositionInfo;
		gShuttleIf[i].Status.ShuttleInfo.Position.Valid := Fbs.ShReadPositionFb[i].Valid;
		gShuttleIf[i].Status.ShuttleInfo.State.Value := Fbs.ShReadState[i].State;
		gShuttleIf[i].Status.ShuttleInfo.State.Valid := Fbs.ShReadState[i].Valid;
	END_FOR;

	IF gAcp6DCtrlIf.Cmd.GetErrorInfo THEN
		Fbs.GetErrorCodesFb.Controller := ADR(gMcAcp6DController);
		Fbs.GetErrorCodesFb.Execute := TRUE;

		IF Fbs.GetErrorCodesFb.Valid OR Fbs.GetErrorCodesFb.Error THEN
			gAcp6DCtrlIf.Status.ErrorCodes := Fbs.GetErrorCodesFb.ErrorCodes;
			Fbs.GetErrorCodesFb.Execute := FALSE;
			gAcp6DCtrlIf.Cmd.GetErrorInfo := FALSE;
		END_IF

	END_IF
	Fbs.CfgReadCyclicPos();
	Fbs.GetErrorCodesFb();
	Fbs.SysReadStateFb();
	Fbs.PowerOffFb();
	Fbs.PowerOnFb();
	Fbs.AutoRefreshFB();

	gAcp6DCtrlIf.Status.Ready := state = ACP6D_READY;
	gAcp6DCtrlIf.Status.Error := state = ACP6D_ERROR;
	gAcp6DCtrlIf.Status.ReadyToPowerOn := Fbs.SysReadStateFb.Valid AND Fbs.SysReadStateFb.State = mcACP6D_STATE_INACTIVE;

END_PROGRAM
```

### Program Logical/Source/6DCtrl/MacroLoad

#### Init.st
```iecst
PROGRAM _INIT
	//Enable the macros for loading
	gMacroLoadIf.Par.MacroList[0].Load := TRUE;
	gMacroLoadIf.Par.MacroList[0].MacroFileName := '128_RobotSyncDemo.xml';
	gMacroLoadIf.Par.MacroList[0].MacroID := 128;

	//Define the parameters for the macro load IF
	gMacroLoadIf.Par.FileDevice := '6DMacro';
END_PROGRAM
```

### Program Logical/Source/Auxil/OeeCalc

#### Variables.var
```iecst
VAR
	SysThroughputCalcFb : ThroughputCounterFb;
END_VAR
```

#### Cyclic.st
```iecst
PROGRAM _CYCLIC

	SysThroughputCalcFb.Enable := gProcessInfoIf.Cmd.Enable;
	SysThroughputCalcFb.ProductCounter := gProcessInfoIf.Par.CurrentProductCount;
	SysThroughputCalcFb.Reset := gProcessInfoIf.Cmd.ResetData;

	gProcessInfoIf.Sts.Enabled := gProcessInfoIf.Cmd.Enable;
	IF gProcessInfoIf.Cmd.ResetData THEN
		gProcessInfoIf.Cmd.ResetData := FALSE;
		gProcessInfoIf.Par.CurrentProductCount := 0;
	END_IF

	SysThroughputCalcFb();

	gProcessInfoIf.Sts.CurrentBlistersPerMinute := SysThroughputCalcFb.PPM * 6;
	gProcessInfoIf.Sts.CurrentLayersPerMinute := SysThroughputCalcFb.PPM * 4;
	gProcessInfoIf.Sts.CurrentPPM := SysThroughputCalcFb.PPM;
	gProcessInfoIf.Sts.CurrentPPH := SysThroughputCalcFb.PPH;
END_PROGRAM
```

### Program Logical/Source/Robot/RbtCtrl (IEC)

#### Types.typ
```iecst
TYPE
	RobotStatesEnum :
		(
		RBT_OFF,
		RBT_POWER_ON,
		RBT_HOME,
		RBT_IDLE,
		RBT_WAITING_TO_SYNC,
		RBT_SYNC,
		RBT_DESYNC,
		RBT_MOVE_TO_SYNC,
		RBT_RUN,
		RBT_ERROR
		);
END_TYPE
```

#### Variables.var
```iecst
VAR
	RoboBasicFb : MpDelta3Axis;
	deltaPars : MpDelta3AxisParType := (ProgramName:='Demo.gcode');
	state : RobotStatesEnum;
	getCoordSystemIdent : MC_BR_GetCoordSystemIdent;
	OnlinePath : MC_BR_OnlinePathInfluence_15;
	masterPositionFb : MC_BR_ReadCyclicPosition;
END_VAR
```

#### Cyclic.st
```iecst
PROGRAM _CYCLIC
	RoboBasicFb.MpLink := ADR(g3AxDeltaA);
	OnlinePath.AxesGroup := ADR(g3AxDeltaA);

	CASE state OF
		RBT_OFF:
			gSceneViewerIf.Cmds.Clear := TRUE;
			gSceneViewerIf.Cmds.Record := FALSE;

			IF gRobotIf.Cmds.Admin.Power THEN
				RoboBasicFb.Power := TRUE;
				gSceneViewerIf.Cmds.Clear := FALSE;
				gSceneViewerIf.Cmds.Record := TRUE;

				state := RBT_POWER_ON;
			END_IF

		RBT_POWER_ON:
			IF RoboBasicFb.PowerOn THEN
				gRobotIf.Status.Powered := TRUE;
			ELSIF NOT gRobotIf.Status.Homed THEN
				RoboBasicFb.Home := TRUE;

				state := RBT_HOME;
			ELSE
				state := RBT_IDLE;
			END_IF

		RBT_HOME:
			IF RoboBasicFb.IsHomed THEN
				gRobotIf.Cmds.Admin.Home := FALSE;
				RoboBasicFb.Home := FALSE;

				gRobotIf.Status.Homed := TRUE;

				state := RBT_IDLE;
			END_IF

		RBT_IDLE:
			IF gRobotIf.Cmds.Admin.Home THEN
				gRobotIf.Status.Homed := FALSE;
				RoboBasicFb.Home := TRUE;

				state := RBT_HOME;
			ELSIF gRobotIf.Cmds.Process.Run THEN
				getCoordSystemIdent.Execute := TRUE;
				getCoordSystemIdent.CoordSystemName := gRobotIf.Pars.SyncFrame;

				getCoordSystemIdent.Parameter.AxesGroup := ADR(g3AxDeltaA);

				getCoordSystemIdent();

				RoboBasicFb.MoveProgram := TRUE;
				IF RoboBasicFb.Info.Program.ProgramPhase = mcPRGPH_REAL_RUN AND getCoordSystemIdent.Done THEN

					gPickPlaceIf.Run := TRUE;
					gRobotIf.Pars.SyncFrameIdent := getCoordSystemIdent.Ident;
					deltaPars.CoordSystem := gRobotIf.Pars.SyncFrameIdent;
					OnlinePath.CoordSystem := deltaPars.CoordSystem;
					getCoordSystemIdent.Execute := FALSE;

					state := RBT_RUN;
				END_IF

			ELSE
				IF(gRobotIf.Cmds.Process.Sync) THEN
					//Get the position
					masterPositionFb.Axis := ADR(gSyncIf.Status.AxisToSync);
					masterPositionFb.Enable := TRUE;

					OnlinePath.Enable := TRUE;

					RoboBasicFb.MoveProgram := TRUE;

					IF(RoboBasicFb.Info.Program.ProgramPhase = mcPRGPH_REAL_RUN AND gRobotIf.Pars.ShuttleIdx <> STATION_IS_EMPTY AND OnlinePath.Enabled) THEN
						OnlinePath.PositionOffset[0] := masterPositionFb.CyclicPosition * 1000 - gRobotIf.Pars.SyncPosition.X;
						gRobotIf.Status.AtSync := FALSE;

						gRobotIf.Status.Synced := TRUE;

						state := RBT_SYNC;
					END_IF
				END_IF
			END_IF

		RBT_MOVE_TO_SYNC:
			IF(RoboBasicFb.MoveDone) THEN
				gRobotIf.Status.AtSync := TRUE;
				RoboBasicFb.MoveDirect := FALSE;

				state := RBT_IDLE;
			END_IF

		RBT_SYNC:
			IF(masterPositionFb.Valid) THEN
				//Continually update the online path influencer with the shuttle's position corrected for the offset
				OnlinePath.PositionOffset[0] := masterPositionFb.CyclicPosition * 1000 - gRobotIf.Pars.SyncPosition.X;
			END_IF

			//Gcode program sets the flag to be false when the "place" or w/e routine has finished. When this happens,
			//	Stop the online path influencer, stop the cyclic pos read, and tell the track to go ahead and release the shuttle
			IF(NOT gPickPlaceIf.Status.ProductPresent) THEN

				gRobotIf.Status.Synced := FALSE;
				gPickPlaceIf.Status.ProductOK := TRUE;
				gSyncIf.Cmds.Proc.ReleaseUnSync := TRUE;

				OnlinePath.Enable := FALSE;
				brsmemset(ADR(OnlinePath.PositionOffset),0,SIZEOF(OnlinePath.PositionOffset));
				masterPositionFb.Enable := FALSE;

				state := RBT_RUN;
			END_IF
		RBT_RUN:
		//Running the program right now
			IF(gSyncIf.Status.SyncReady AND gPickPlaceIf.Status.ProductPresent) THEN
				masterPositionFb.Axis := ADR(gSyncIf.Status.AxisToSync);
				masterPositionFb.Enable := TRUE;
				gRobotIf.Status.Synced := TRUE;
				gPickPlaceIf.Sync := TRUE;

				//Tell the Trak to release the shuttle
				gSyncIf.Cmds.Proc.ReleaseSync := TRUE;
				OnlinePath.Enable := TRUE;

				state := RBT_SYNC;
			END_IF

		END_CASE

		RoboBasicFb();
		OnlinePath();
		masterPositionFb();

END_PROGRAM
```

#### Exit.st
```iecst
PROGRAM _EXIT
	RoboBasicFb.Enable := FALSE;
	RoboBasicFb();

END_PROGRAM
```

#### Init.st
```iecst
PROGRAM _INIT
	RoboBasicFb.Enable := TRUE;
	RoboBasicFb.MpLink := ADR(g3AxDeltaA);
	RoboBasicFb.Override := 100;
	RoboBasicFb.Parameters := ADR(deltaPars);

	RoboBasicFb();

	brsstrcpy(ADR(gRobotIf.Pars.SyncFrame),ADR("TrakSync"));
	gRobotIf.Pars.SyncPosition.X := 150;
	gRobotIf.Pars.SyncPosition.Y := 0;
	gRobotIf.Pars.SyncPosition.Z := 0;
	gRobotIf.Pars.MoveToSyncVel := 700;
	gRobotIf.Pars.MoveToSyncAccel := 2000;
	gRobotIf.Pars.MoveToSyncDecel := 2000;

	//Setting these in the TrakSyncframe!!
	gPickPlaceIf.Config.PickLoc.X := 330;
	gPickPlaceIf.Config.PickLoc.Y := -200;
	gPickPlaceIf.Config.PickLoc.Z := 50;

	gPickPlaceIf.Config.PlaceLoc.X := 150;
	gPickPlaceIf.Config.PlaceLoc.Y := 0;
	gPickPlaceIf.Config.PlaceLoc.Z := 0;

	gPickPlaceIf.Pars.PickTune.ApproachHeight := 50;
	gPickPlaceIf.Pars.PickTune.DepartHeight := 30;
	gPickPlaceIf.Pars.PickTune.Radius := 40;
	gPickPlaceIf.Pars.PickTune.DwellTime := 0.10;

	gPickPlaceIf.Pars.ProductSpeed.Vel := 250;
	gPickPlaceIf.Pars.ProductSpeed.Accel := 1000;
	gPickPlaceIf.Pars.ProductSpeed.Decel := 1000;

	gPickPlaceIf.Pars.EmptySpeed.Vel := 500;
	gPickPlaceIf.Pars.EmptySpeed.Accel := 2000;
	gPickPlaceIf.Pars.EmptySpeed.Decel := 2000;

END_PROGRAM
```

### Program Logical/Source/Demos/MacroDemo (IEC)

#### Types.typ
```iecst
TYPE
	MacroDemoStateEnum :
		(
		MD_IDLE,
		MD_LOAD_FILE,
		MD_RUN_MACRO,
		MD_DONE,
		MD_RESET,
		MD_ERROR
		);
	MacroDemoModeEnum :
		(
		mdFILE,
		mdID
		);
	MacroDemoIfTyp : 	STRUCT
		Cmd : MacroDemoCmdTyp;
		Cfg : MacroDemoCfgTyp;
		Par : MacroDemoParTyp;
		Sts : MacroDemoStsTyp;
	END_STRUCT;
	MacroDemoCmdTyp : 	STRUCT
		Run : BOOL;
		Reset : BOOL;
	END_STRUCT;
	MacroDemoCfgTyp : 	STRUCT
		FileDevice : STRING[80];
	END_STRUCT;
	MacroDemoParTyp : 	STRUCT
		ShId : USINT;
		MacroId : USINT;
		MacroFileName : STRING[80];
		Mode : MacroDemoModeEnum;
	END_STRUCT;
	MacroDemoStsTyp : 	STRUCT
		Running : BOOL;
		Error : BOOL;
	END_STRUCT;
	MacroDemoFbsTyp : 	STRUCT
		LoadMacroFb : MC_BR_MacroLoad_Acp6D;
		RunMacroFb : MC_BR_MacroRun_Acp6D;
	END_STRUCT;
END_TYPE
```

#### Variables.var
```iecst
VAR
	state : MacroDemoStateEnum;
	macroDemoIf : MacroDemoIfTyp;
	demoFbs : MacroDemoFbsTyp;
END_VAR
```

#### Cyclic.st
```iecst
(*
	This demo connects to the HMI to run pre configured macros on shuttles. Move the shuttle in the desired starting position BEFORE executing the demo (or ensure the macro moves the shuttle to the desired starting location)
*)
PROGRAM _CYCLIC
	//Steps

	(*
		Wait for a command to execute
			If in FileMode, load the defined macro on to the controller
			If not, execute the macro on the defined shuttle
		Macro Load
			when completed, exectue the macro on the defined shuttle
		Macro Run
			When acknowledged, head to the done state
		Done
			When cmd dropped, move to reset
		Reset
			Reset all bits and head back to the idle state
		Error
			wait for a reset command and then move to the reset state

	*)

	CASE state OF
		MD_IDLE://******************************************************************************** Idle state waiting for a command
			IF macroDemoIf.Cmd.Run THEN
				demoFbs.LoadMacroFb.Controller := ADR(gMcAcp6DController);
				demoFbs.RunMacroFb.Controller := ADR(gMcAcp6DController);
				demoFbs.RunMacroFb.ShuttleID := macroDemoIf.Par.ShId;

				CASE macroDemoIf.Par.Mode OF
					mdFILE:
						state := MD_LOAD_FILE;
					mdID:
						state := MD_RUN_MACRO;
				END_CASE;
			END_IF
		MD_LOAD_FILE://******************************************************************************** Demo is loading the defined file
			demoFbs.LoadMacroFb.FileDevice := macroDemoIf.Cfg.FileDevice;
			demoFbs.LoadMacroFb.FileName := macroDemoIf.Par.MacroFileName;
			demoFbs.LoadMacroFb.MacroID := macroDemoIf.Par.MacroId;
			demoFbs.LoadMacroFb.Execute := TRUE;

			IF demoFbs.LoadMacroFb.Error THEN
				macroDemoIf.Sts.Error := TRUE;

				state := MD_ERROR;
			ELSIF demoFbs.LoadMacroFb.Done THEN
				demoFbs.LoadMacroFb.Execute := FALSE;

				state := MD_RUN_MACRO;
			END_IF

		MD_RUN_MACRO://******************************************************************************** Demo is running the defined macro
			demoFbs.RunMacroFb.MacroID := macroDemoIf.Par.MacroId;
			demoFbs.RunMacroFb.Execute := TRUE;

			IF demoFbs.RunMacroFb.Error THEN
				macroDemoIf.Sts.Error := TRUE;

				state := MD_ERROR;
			ELSIF demoFbs.RunMacroFb.Acknowledge THEN
				demoFbs.RunMacroFb.Execute := FALSE;

				state := MD_DONE;
			END_IF
		MD_DONE://******************************************************************************** Demo has compelted
			state := MD_RESET;
		MD_RESET://******************************************************************************** Demo resetting all values/variables/fbs
			macroDemoIf.Cmd.Run := FALSE;
			macroDemoIf.Cmd.Reset := FALSE;

			demoFbs.RunMacroFb.Execute := FALSE;
			demoFbs.LoadMacroFb.Execute := FALSE;

			macroDemoIf.Sts.Error := FALSE;
			macroDemoIf.Sts.Running := FALSE;

			state := MD_IDLE;
		MD_ERROR://******************************************************************************** Demo in error state
			IF macroDemoIf.Cmd.Reset THEN
				state := MD_RESET;
			END_IF
	END_CASE;

	demoFbs.LoadMacroFb();
	demoFbs.RunMacroFb();
END_PROGRAM
```

#### Init.st
```iecst
PROGRAM _INIT
	macroDemoIf.Cfg.FileDevice := '6DMacro';

END_PROGRAM
```

### Program Logical/Source/Demos/VariedMovDemo (IEC)

#### LocalFunctionsTypes.typ
```iecst
(*Angled Movement Function block*)

TYPE
	AngledMovementInternalTyp : 	STRUCT
		state : AngledMovementInternalStateEnum;
		Fbs : AngledMovementInternalFbsTyp;
		ShPos : ARRAY[0..5]OF REAL;
		MovementNum : USINT;
	END_STRUCT;
	AngledMovementInternalFbsTyp : 	STRUCT
		Move6DFb : MC_BR_Move6D_Acp6D;
	END_STRUCT;
	AngledMovementInternalStateEnum :
		(
		ANG_INT_OFF,
		ANG_INT_MOV_WAIT,
		ANG_INT_MOV_1,
		ANG_INT_MOV_2,
		ANG_INT_MOV_3,
		ANG_INT_MOV_4,
		ANG_INT_MOV_5,
		ANG_INT_MOV_6,
		ANG_INT_MOV_7,
		ANG_INT_MOV_8,
		ANG_INT_MOV_9,
		ANG_INT_MOV_10,
		ANG_INT_DONE,
		ANG_INT_RESET,
		ANG_INT_ERROR
		);
END_TYPE

(*"wobble movement function block"*)

TYPE
	WobbleMovInternalTyp : 	STRUCT
		state : WobbleMovStateEnum;
		Fbs : WobbleMovInternalFbsTyp;
	END_STRUCT;
	WobbleMovInternalFbsTyp : 	STRUCT
		VirtualMacroFb : MC_BR_MacroRun_Acp6D;
		RealMacroFb : MC_BR_MacroRun_Acp6D;
		PlanetCtrlFb : MC_BR_PlanetCtrl_Acp6D;
		StopFb : MC_BR_Stop_Acp6D;
		Move6DFb : MC_BR_Move6D_Acp6D;
	END_STRUCT;
	WobbleMovStateEnum :
		(
		WOB_INT_OFF,
		WOB_INT_SETUP_PLANET,
		WOB_INT_MACRO_RUN,
		WOB_INT_STOP,
		WOB_INT_REORIENT,
		WOB_INT_BREAK_PLANET,
		WOB_INT_RESET,
		WOB_INT_DONE,
		WOB_INT_ERROR
		);
END_TYPE
```

#### Types.typ
```iecst
TYPE
	FillStationStateEnum :
		(
		FILL_OFF, (*Fill station is currently disabled*)
		FILL_INIT, (*Fill station is initalizing*)
		FILL_WAIT_FOR_SHUTTLE, (*Fill station is waiting for a shuttle to be present*)
		FILL_ENTER_SHUTTLE, (*Shuttle is entering the filling station*)
		FILL_FILLING, (*Fill station is preforming the filling process*)
		FILL_EXIT_SHUTTLE, (*Fill station is preforming the exit movement*)
		FILL_DONE, (*Fill station is done with the filling process*)
		FILL_CHECK_REPEAT,
		FILL_RESET,
		FILL_ERROR (*Fill station had an error*)
		);
	FillStationFbTyp : 	STRUCT
		FillMoveFb : MC_BR_MoveInPlane_Acp6D;
		WaitTimer : TON;
		St1Fb : AngledMovementFb;
		St2Fb : MC_BR_MacroRun_Acp6D;
		St3Fb : WobbleMovementFb;
		St4Fb : MC_BR_MacroRun_Acp6D;
	END_STRUCT;
	FillStationParsTyp : 	STRUCT
		Vel : REAL;
		Accel : REAL;
		FillRate : REAL;
		FillTime : TIME;
		RepeatLimit : USINT;
		Repeat : BOOL;
	END_STRUCT;
END_TYPE
```

#### Variables.var
```iecst
VAR
	state : ARRAY[0..1] OF FillStationStateEnum;
	stationFbs : ARRAY[0..1] OF FillStationFbTyp;
	taskName : STRING[80];
	stationPars : {REDUND_UNREPLICABLE} FillStationParsTyp;
	station : FillStationEnum;
	macroPatternCounter : ARRAY[0..1] OF USINT;
	repeatCounter : USINT;
	i : INT;
END_VAR
```

#### LocalFunctions.fun
```iecst
{REDUND_ERROR} FUNCTION_BLOCK AngledMovementFb (*TODO: Add your comment here*) (*$GROUP=User,$CAT=User,$GROUPICON=User.png,$CATICON=User.png*)
	VAR_INPUT
		Execute : BOOL;
		Reset : BOOL;
		Controller : REFERENCE TO McAcp6DControllerType;
		ShuttleId : USINT;
		PosStartX : REAL;
		PosStartY : REAL;
		LinearVel : REAL;
		ShortAxisRotVel : REAL;
	END_VAR
	VAR_OUTPUT
		Active : BOOL;
		Done : BOOL;
		Error : BOOL;
	END_VAR
	VAR
		Internal : AngledMovementInternalTyp;
	END_VAR
END_FUNCTION_BLOCK

{REDUND_ERROR} FUNCTION_BLOCK WobbleMovementFb (*TODO: Add your comment here*) (*$GROUP=User,$CAT=User,$GROUPICON=User.png,$CATICON=User.png*)
	VAR_INPUT
		Execute : BOOL;
		Reset : BOOL;
		Controller : REFERENCE TO McAcp6DControllerType;
		ShuttleId : USINT;
		VirtShId : USINT;
		SunMacroID : USINT;
		PlanetMacroID : USINT;
		PosStartX : REAL;
		PosStartY : REAL;
	END_VAR
	VAR_OUTPUT
		Active : BOOL;
		Done : BOOL;
		Error : BOOL;
	END_VAR
	VAR
		Internal : WobbleMovInternalTyp;
	END_VAR
END_FUNCTION_BLOCK
```

#### AngledMovementFb.st
```iecst
FUNCTION_BLOCK AngledMovementFb
	IF Reset THEN
		Internal.state := ANG_INT_RESET;
	END_IF
	CASE Internal.state OF
		ANG_INT_OFF:
			IF Execute THEN
				Active := TRUE;
				Internal.ShPos[axPosX] := PosStartX - 0.026;
				Internal.ShPos[axPosY] := PosStartY + 0.026;
				Internal.ShPos[axPosZ] := 0.003;
				Internal.ShPos[axPosRX] := 0.02;
				Internal.ShPos[axPosRY] := 0.02;

				Internal.Fbs.Move6DFb.Controller := ADR(Controller);
				Internal.Fbs.Move6DFb.ShuttleID := ShuttleId;
				Internal.Fbs.Move6DFb.Position := Internal.ShPos;
				Internal.Fbs.Move6DFb.InPlaneVelocity := LinearVel;
				Internal.Fbs.Move6DFb.Acceleration := 10;
				Internal.Fbs.Move6DFb.ShortAxisVelocity[axVel] := LinearVel;
				Internal.Fbs.Move6DFb.ShortAxisVelocity[axVelRx] := ShortAxisRotVel;
				Internal.Fbs.Move6DFb.ShortAxisVelocity[axVelRy] := ShortAxisRotVel;
				Internal.Fbs.Move6DFb.ShortAxisVelocity[axVelRz] := ShortAxisRotVel;

				Internal.Fbs.Move6DFb.Execute := TRUE;

				Internal.state := ANG_INT_MOV_WAIT;
			END_IF
		ANG_INT_MOV_WAIT:
			IF Internal.Fbs.Move6DFb.Done THEN
				Internal.Fbs.Move6DFb.Execute := FALSE;
				Internal.MovementNum := Internal.MovementNum + 1;
				IF Internal.MovementNum >= 11 THEN
					Done := TRUE;
					Internal.state := ANG_INT_DONE;
				ELSE
					Internal.state := ANG_INT_MOV_WAIT + Internal.MovementNum;
				END_IF

			END_IF
		ANG_INT_MOV_1:
			Internal.ShPos[axPosX] := Internal.ShPos[axPosX];
			Internal.ShPos[axPosY] := Internal.ShPos[axPosY] - 0.052;
			Internal.ShPos[axPosRX] := -0.02;
			Internal.ShPos[axPosRY] := 0.02;

			Internal.Fbs.Move6DFb.Position := Internal.ShPos;
			Internal.Fbs.Move6DFb.Execute := TRUE;

			Internal.state := ANG_INT_MOV_WAIT;
		ANG_INT_MOV_2:
			Internal.ShPos[axPosX] := Internal.ShPos[axPosX] + 0.052;
			Internal.ShPos[axPosY] := Internal.ShPos[axPosY];
			Internal.ShPos[axPosRX] := -0.02;
			Internal.ShPos[axPosRY] := -0.02;

			Internal.Fbs.Move6DFb.Position := Internal.ShPos;
			Internal.Fbs.Move6DFb.Execute := TRUE;

			Internal.state := ANG_INT_MOV_WAIT;
		ANG_INT_MOV_3:
			Internal.ShPos[axPosX] := Internal.ShPos[axPosX];
			Internal.ShPos[axPosY] := Internal.ShPos[axPosY] + 0.052;
			Internal.ShPos[axPosRX] := 0.02;
			Internal.ShPos[axPosRY] := -0.02;

			Internal.Fbs.Move6DFb.Position := Internal.ShPos;
			Internal.Fbs.Move6DFb.Execute := TRUE;

			Internal.state := ANG_INT_MOV_WAIT;
		ANG_INT_MOV_4:
			Internal.ShPos[axPosX] := Internal.ShPos[axPosX] - 0.052;
			Internal.ShPos[axPosY] := Internal.ShPos[axPosY];
			Internal.ShPos[axPosRX] := 0.02;
			Internal.ShPos[axPosRY] := 0.02;

			Internal.Fbs.Move6DFb.Position := Internal.ShPos;
			Internal.Fbs.Move6DFb.Execute := TRUE;

			Internal.state := ANG_INT_MOV_WAIT;
		ANG_INT_MOV_5:
			Internal.ShPos[axPosX] := Internal.ShPos[axPosX] + 0.015;
			Internal.ShPos[axPosY] := Internal.ShPos[axPosY] - 0.015;
			Internal.ShPos[axPosRX] := 0.0;
			Internal.ShPos[axPosRY] := 0.0;

			Internal.Fbs.Move6DFb.Position := Internal.ShPos;
			Internal.Fbs.Move6DFb.Execute := TRUE;

			Internal.state := ANG_INT_MOV_WAIT;
		ANG_INT_MOV_6:
			Internal.ShPos[axPosX] := Internal.ShPos[axPosX];
			Internal.ShPos[axPosY] := Internal.ShPos[axPosY] - 0.026;
			Internal.ShPos[axPosRX] := 0.0;
			Internal.ShPos[axPosRY] := 0.0;

			Internal.Fbs.Move6DFb.Position := Internal.ShPos;
			Internal.Fbs.Move6DFb.Execute := TRUE;

			Internal.state := ANG_INT_MOV_WAIT;
		ANG_INT_MOV_7:
			Internal.ShPos[axPosX] := Internal.ShPos[axPosX] + 0.026;
			Internal.ShPos[axPosY] := Internal.ShPos[axPosY];
			Internal.ShPos[axPosRX] := 0.0;
			Internal.ShPos[axPosRY] := 0.0;

			Internal.Fbs.Move6DFb.Position := Internal.ShPos;
			Internal.Fbs.Move6DFb.Execute := TRUE;

			Internal.state := ANG_INT_MOV_WAIT;
		ANG_INT_MOV_8:
			Internal.ShPos[axPosX] := Internal.ShPos[axPosX];
			Internal.ShPos[axPosY] := Internal.ShPos[axPosY] + 0.026;
			Internal.ShPos[axPosRX] := 0.0;
			Internal.ShPos[axPosRY] := 0.0;

			Internal.Fbs.Move6DFb.Position := Internal.ShPos;
			Internal.Fbs.Move6DFb.Execute := TRUE;

			Internal.state := ANG_INT_MOV_WAIT;
		ANG_INT_MOV_9:
			Internal.ShPos[axPosX] := Internal.ShPos[axPosX] - 0.026;
			Internal.ShPos[axPosY] := Internal.ShPos[axPosY];
			Internal.ShPos[axPosRX] := 0.0;
			Internal.ShPos[axPosRY] := 0.0;

			Internal.Fbs.Move6DFb.Position := Internal.ShPos;
			Internal.Fbs.Move6DFb.Execute := TRUE;

			Internal.state := ANG_INT_MOV_WAIT;
		ANG_INT_MOV_10:
			Internal.ShPos[axPosX] := PosStartX;
			Internal.ShPos[axPosY] := PosStartY;
			Internal.ShPos[axPosZ] := 0.002;
			Internal.ShPos[axPosRX] := 0.0;
			Internal.ShPos[axPosRY] := 0.0;

			Internal.Fbs.Move6DFb.Position := Internal.ShPos;
			Internal.Fbs.Move6DFb.Execute := TRUE;

			Internal.state := ANG_INT_MOV_WAIT;

		ANG_INT_DONE:
			IF NOT Execute THEN
				Internal.state := ANG_INT_RESET;
			END_IF
		ANG_INT_RESET:
			Internal.Fbs.Move6DFb.Execute := FALSE;
			Execute := FALSE;
			Reset := FALSE;
			Internal.MovementNum := 0;

			Active := FALSE;
			Done := FALSE;
			Error := FALSE;

			Internal.state := ANG_INT_OFF;
		ANG_INT_ERROR:
			IF NOT Execute OR Reset THEN
				Internal.state := ANG_INT_RESET;
			END_IF
	END_CASE;
	Internal.Fbs.Move6DFb();
END_FUNCTION_BLOCK
```

#### Cyclic.st
```iecst
PROGRAM _CYCLIC
	FOR i:=0 TO 1 DO
		CASE state[i] OF
			FILL_OFF: //********************************************************************************Fill station is currently disabled
				IF gVariedMoveDemoIf[i].Cmd.Enable THEN
					state[i] := FILL_INIT;
				END_IF
			FILL_INIT: //********************************************************************************Fill station is initalizing
				gVariedMoveDemoIf[i].Sts.ReadyForNewShuttle := TRUE;
				gVariedMoveDemoIf[i].Sts.Enabled := TRUE;
				state[i] := FILL_WAIT_FOR_SHUTTLE;
			FILL_WAIT_FOR_SHUTTLE: //********************************************************************************Fill station is waiting for a shuttle to be present
				IF NOT gVariedMoveDemoIf[i].Cmd.Enable THEN
					gVariedMoveDemoIf[i].Sts.ReadyForNewShuttle := FALSE;
					gVariedMoveDemoIf[i].Sts.Enabled := FALSE;
					state[i] := FILL_OFF;
				ELSIF gVariedMoveDemoIf[i].Par.ShuttleIdx <> STATION_IS_EMPTY AND gVariedMoveDemoIf[i].Cmd.Process THEN
					gVariedMoveDemoIf[i].Sts.ReadyForNewShuttle := FALSE;
					gVariedMoveDemoIf[i].Sts.Processing := TRUE;

					SetupStationActions;

					state[i] := FILL_FILLING;
				END_IF
			FILL_ENTER_SHUTTLE: //******************************************************************************** Fill station is moving to the filling position
				IF stationFbs[i].FillMoveFb.Error THEN
					gVariedMoveDemoIf[i].Sts.Error := TRUE;

					state[i] := FILL_ERROR;
				ELSIF stationFbs[i].FillMoveFb.Done THEN
					stationFbs[i].FillMoveFb.Execute:= FALSE;

					stationFbs[i].WaitTimer.IN := TRUE;
					stationFbs[i].WaitTimer.PT := stationPars.FillTime;

					SetupStationActions;

					state[i] := FILL_FILLING;
				END_IF
			FILL_FILLING: //********************************************************************************Fill station is preforming the filling process
				IF ((stationFbs[i].St1Fb.Done AND stationFbs[i].St1Fb.Execute)
					OR (stationFbs[i].St2Fb.Done AND stationFbs[i].St2Fb.Execute)
					OR (stationFbs[i].St3Fb.Done AND stationFbs[i].St3Fb.Execute)
					OR (stationFbs[i].St4Fb.Done AND stationFbs[i].St4Fb.Execute)) THEN

					//Interface with the correct Station FB
					CASE gVariedMoveDemoIf[i].Par.StationType OF
						ST1:
							stationFbs[i].St1Fb.Execute := FALSE;
						ST2:
							stationFbs[i].St2Fb.Execute := FALSE;
						ST3:
							stationFbs[i].St3Fb.Execute := FALSE;
							macroPatternCounter[i] := macroPatternCounter[i]+ 1;
							IF macroPatternCounter[i] = 2 THEN
								macroPatternCounter[i] := 0;
							END_IF
						ST4:
							stationFbs[i].St4Fb.Execute := FALSE;
					END_CASE;

					gVariedMoveDemoIf[i].Sts.Done := TRUE;
					gVariedMoveDemoIf[i].Sts.Processing := FALSE;

					state[i] := FILL_DONE;
				END_IF

			FILL_DONE: //********************************************************************************Fill station is done with the load process
				IF NOT gVariedMoveDemoIf[i].Cmd.Enable THEN
					gVariedMoveDemoIf[i].Sts.Enabled := FALSE;
					gVariedMoveDemoIf[i].Sts.ReadyForNewShuttle := FALSE;
					macroPatternCounter[i] := 0;

					state[i] := FILL_RESET;
				ELSE
					gVariedMoveDemoIf[i].Cmd.Process := FALSE;

					gVariedMoveDemoIf[i].Sts.Done := FALSE;
					state[i] := FILL_CHECK_REPEAT;
				END_IF
			FILL_CHECK_REPEAT:
				gVariedMoveDemoIf[i].Sts.RepeatCounter := (gVariedMoveDemoIf[i].Sts.RepeatCounter + 1) * BOOL_TO_USINT(NOT gVariedMoveDemoIf[i].Par.RepeatForever);
				IF gVariedMoveDemoIf[i].Sts.RepeatCounter < gVariedMoveDemoIf[i].Par.RepeatCount OR gVariedMoveDemoIf[i].Par.RepeatForever THEN
					SetupStationActions;
					state[i] := FILL_FILLING;
				ELSE
					gVariedMoveDemoIf[i].Sts.RepeatCounter := 0;
					gVariedMoveDemoIf[i].Par.ShuttleIdx := STATION_IS_EMPTY;
					gVariedMoveDemoIf[i].Sts.ReadyForNewShuttle := FALSE;
					gVariedMoveDemoIf[i].Sts.ReadyForNewShuttle := TRUE;

					state[i] := FILL_WAIT_FOR_SHUTTLE;
				END_IF
			FILL_RESET: //********************************************************************************Reset State
				gVariedMoveDemoIf[i].Cmd.Reset := FALSE;

				gVariedMoveDemoIf[i].Sts.Done := FALSE;
				gVariedMoveDemoIf[i].Sts.Error := FALSE;
				gVariedMoveDemoIf[i].Sts.Processing := FALSE;
				gVariedMoveDemoIf[i].Sts.ReadyForNewShuttle := FALSE;
				gVariedMoveDemoIf[i].Sts.Enabled := FALSE;

				stationFbs[i].FillMoveFb.Execute := FALSE;
				stationFbs[i].WaitTimer.IN := FALSE;
				IF gVariedMoveDemoIf[i].Cmd.Enable THEN
					state[i] := FILL_INIT;
				ELSE
					state[i] := FILL_OFF;
				END_IF
			FILL_ERROR: //********************************************************************************Fill station had an error
				IF gVariedMoveDemoIf[i].Cmd.Reset THEN
					state[i] := FILL_RESET;
				END_IF
		END_CASE;

		stationFbs[i].FillMoveFb();
		stationFbs[i].WaitTimer();
		//Call the appropriate station block
		CallStationFbs;

	END_FOR;

END_PROGRAM
```

#### Init.st
```iecst
PROGRAM _INIT
	station := ST1;

	gVariedMoveDemoIf[0].Par.StationType := ST1;
	gVariedMoveDemoIf[0].Cmd.Enable := TRUE;
	gVariedMoveDemoIf[0].Cfg.StationPos.X := 0.12;
	gVariedMoveDemoIf[0].Cfg.StationPos.Y := 0.12;
	gVariedMoveDemoIf[1].Par.StationType := ST2;
	gVariedMoveDemoIf[1].Cmd.Enable := TRUE;
	gVariedMoveDemoIf[1].Cfg.StationPos.X := 0.36;
	gVariedMoveDemoIf[1].Cfg.StationPos.Y := 0.12;

	stationPars.Vel := 1.0;
	stationPars.Accel := 10.0;

	stationFbs[0].St1Fb.LinearVel := 0.5;// m/s
	stationFbs[0].St1Fb.ShortAxisRotVel := 0.5;//rad/s
	stationFbs[1].St1Fb.LinearVel := 0.5;// m/s
	stationFbs[1].St1Fb.ShortAxisRotVel := 0.5;//rad/s
END_PROGRAM
```

#### StationActions.st
```iecst
ACTION SetupStationActions:
	CASE gVariedMoveDemoIf[i].Par.StationType OF
		ST1:
			stationFbs[i].St1Fb.Execute := TRUE;
			stationFbs[i].St1Fb.Controller := ADR(gMcAcp6DController);
			stationFbs[i].St1Fb.ShuttleId := gShuttleIf[gVariedMoveDemoIf[i].Par.ShuttleIdx].Cfg.ShuttleId;
			stationFbs[i].St1Fb.PosStartX := gVariedMoveDemoIf[i].Cfg.StationPos.X;
			stationFbs[i].St1Fb.PosStartY := gVariedMoveDemoIf[i].Cfg.StationPos.Y;
		ST2:
			stationFbs[i].St2Fb.Controller := ADR(gMcAcp6DController);
			stationFbs[i].St2Fb.MacroID := DINT_TO_USINT(140);
			stationFbs[i].St2Fb.ShuttleID := gShuttleIf[gVariedMoveDemoIf[i].Par.ShuttleIdx].Cfg.ShuttleId;
			stationFbs[i].St2Fb.Execute := TRUE;
		ST3:
			stationFbs[i].St3Fb.Controller := ADR(gMcAcp6DController);
			stationFbs[i].St3Fb.PosStartX := gVariedMoveDemoIf[i].Cfg.StationPos.X;
			stationFbs[i].St3Fb.PosStartY := gVariedMoveDemoIf[i].Cfg.StationPos.Y;
			stationFbs[i].St3Fb.PlanetMacroID := DINT_TO_USINT(142);

			stationFbs[i].St3Fb.ShuttleId := gShuttleIf[gVariedMoveDemoIf[i].Par.ShuttleIdx].Cfg.ShuttleId;
			stationFbs[i].St3Fb.VirtShId := 100 + INT_TO_USINT(i);
			stationFbs[i].St3Fb.Execute := TRUE;
			stationFbs[i].St3Fb.SunMacroID := DINT_TO_USINT(141);
			CASE macroPatternCounter[i] OF
				0:
					stationFbs[i].St3Fb.SunMacroID := DINT_TO_USINT(141);
				1:
					stationFbs[i].St3Fb.SunMacroID := DINT_TO_USINT(170);
				2:
					stationFbs[i].St3Fb.SunMacroID := DINT_TO_USINT(171);
			END_CASE;

		ST4:
			stationFbs[i].St4Fb.Controller := ADR(gMcAcp6DController);
			stationFbs[i].St4Fb.MacroID := DINT_TO_USINT(143);
			stationFbs[i].St4Fb.ShuttleID := gShuttleIf[gVariedMoveDemoIf[i].Par.ShuttleIdx].Cfg.ShuttleId;
			stationFbs[i].St4Fb.Execute := TRUE;
	END_CASE;
END_ACTION

ACTION CallStationFbs:
	CASE gVariedMoveDemoIf[i].Par.StationType OF
		ST1:
			stationFbs[i].St1Fb();
		ST2:
			stationFbs[i].St2Fb();
		ST3:
			stationFbs[i].St3Fb();
		ST4:
			stationFbs[i].St4Fb();
	END_CASE;
END_ACTION
```

#### WobbleMovementFb.st
```iecst
FUNCTION_BLOCK WobbleMovementFb
	//Setup Sun/Planet
	//Run Macro on Virtual
	//Run Wobble Macro on Real
	//When Virtual macro finishes, issue stop command to Real
	//Move6D to real shuttle
	//Exit Sun/Planet
	IF Reset THEN
		Internal.state := WOB_INT_RESET;
	END_IF
	CASE Internal.state OF
		WOB_INT_OFF:
			IF Execute THEN
				Active := TRUE;

				Internal.Fbs.PlanetCtrlFb.Controller := ADR(Controller);
				Internal.Fbs.PlanetCtrlFb.NumberOfPlanets := 1;
				Internal.Fbs.PlanetCtrlFb.PlanetShuttleID[0] := ShuttleId;
				Internal.Fbs.PlanetCtrlFb.StarShuttleID := VirtShId;
				Internal.Fbs.PlanetCtrlFb.Level := mcACP6D_PLANET_CONNECT;
				Internal.Fbs.PlanetCtrlFb.Execute := TRUE;

				Internal.state := WOB_INT_SETUP_PLANET;
			END_IF
		WOB_INT_SETUP_PLANET:
			IF Internal.Fbs.PlanetCtrlFb.Error THEN
				Internal.state := WOB_INT_ERROR;
			ELSIF Internal.Fbs.PlanetCtrlFb.Done THEN
				Internal.Fbs.PlanetCtrlFb.Execute := FALSE;

				Internal.Fbs.VirtualMacroFb.Controller := ADR(Controller);
				Internal.Fbs.VirtualMacroFb.MacroID := SunMacroID;
				Internal.Fbs.VirtualMacroFb.ShuttleID := VirtShId;
				Internal.Fbs.VirtualMacroFb.Execute := TRUE;

				Internal.Fbs.RealMacroFb.Controller := ADR(Controller);
				Internal.Fbs.RealMacroFb.MacroID := PlanetMacroID;
				Internal.Fbs.RealMacroFb.ShuttleID := ShuttleId;
				Internal.Fbs.RealMacroFb.Execute := TRUE;

				Internal.state := WOB_INT_MACRO_RUN;
			END_IF
		WOB_INT_MACRO_RUN:
			IF Internal.Fbs.RealMacroFb.Error OR Internal.Fbs.VirtualMacroFb.Error THEN
				Internal.state := WOB_INT_ERROR;
			ELSIF Internal.Fbs.VirtualMacroFb.Done THEN
				Internal.Fbs.VirtualMacroFb.Execute := FALSE;
				Internal.Fbs.RealMacroFb.Execute := FALSE;

				Internal.Fbs.StopFb.Controller := ADR(Controller);
				Internal.Fbs.StopFb.ShuttleID := ShuttleId;
				Internal.Fbs.StopFb.Execute := TRUE;

				Internal.state := WOB_INT_STOP;
			END_IF
		WOB_INT_STOP:
			IF Internal.Fbs.StopFb.Error THEN
				Internal.state := WOB_INT_ERROR;
			ELSIF Internal.Fbs.StopFb.Done THEN
				Internal.Fbs.StopFb.Execute := FALSE;

				Internal.Fbs.Move6DFb.Controller := ADR(Controller);
				Internal.Fbs.Move6DFb.ShuttleID := ShuttleId;
				Internal.Fbs.Move6DFb.Position[axPosX] := PosStartX;
				Internal.Fbs.Move6DFb.Position[axPosY] := PosStartY;
				Internal.Fbs.Move6DFb.Position[axPosZ] := 0.002;
				Internal.Fbs.Move6DFb.Position[axPosRX] := 0;
				Internal.Fbs.Move6DFb.Position[axPosRY] := 0;
				Internal.Fbs.Move6DFb.Position[axPosRZ] := 0;
				Internal.Fbs.Move6DFb.InPlaneVelocity := 1;
				Internal.Fbs.Move6DFb.Acceleration := 10;
				Internal.Fbs.Move6DFb.ShortAxisVelocity[axVel] := 1;
				Internal.Fbs.Move6DFb.ShortAxisVelocity[axVelRx] := 0.1;
				Internal.Fbs.Move6DFb.ShortAxisVelocity[axVelRy] := 0.1;
				Internal.Fbs.Move6DFb.ShortAxisVelocity[axVelRz] := 0.1;
				Internal.Fbs.Move6DFb.Execute := TRUE;

				Internal.state := WOB_INT_REORIENT;
			END_IF
		WOB_INT_REORIENT:
			IF Internal.Fbs.Move6DFb.Done THEN
				Internal.Fbs.Move6DFb.Execute := FALSE;

				Internal.Fbs.PlanetCtrlFb.Level := mcACP6D_PLANET_DISCONNECT;
				Internal.Fbs.PlanetCtrlFb.Execute := TRUE;

				Internal.state := WOB_INT_BREAK_PLANET;
			END_IF
		WOB_INT_BREAK_PLANET:
			IF Internal.Fbs.PlanetCtrlFb.Error THEN
				Internal.state := WOB_INT_ERROR;
			ELSIF Internal.Fbs.PlanetCtrlFb.Done THEN
				Internal.Fbs.PlanetCtrlFb.Execute := FALSE;
				Done := TRUE;

				Internal.state := WOB_INT_DONE;
			END_IF
		WOB_INT_DONE:
			IF NOT Execute THEN
				Internal.state := WOB_INT_RESET;
			END_IF
		WOB_INT_RESET:
			Internal.Fbs.PlanetCtrlFb.Execute := FALSE;
			Internal.Fbs.RealMacroFb.Execute := FALSE;
			Internal.Fbs.VirtualMacroFb.Execute := FALSE;
			Internal.Fbs.StopFb.Execute := FALSE;
			Internal.Fbs.Move6DFb.Execute := FALSE;

			Active := FALSE;
			Done := FALSE;
			Error := FALSE;

			Internal.state := WOB_INT_OFF;
		WOB_INT_ERROR:
			IF NOT Execute THEN
				Internal.state := WOB_INT_RESET;
			END_IF
	END_CASE;
	Internal.Fbs.PlanetCtrlFb();
	Internal.Fbs.RealMacroFb();
	Internal.Fbs.VirtualMacroFb();
	Internal.Fbs.StopFb();
	Internal.Fbs.Move6DFb();
END_FUNCTION_BLOCK
```

### Program Logical/Source/Demos/ConvUnload (IEC)

#### Types.typ
```iecst
TYPE
	ConvHandOffIfTyp : 	STRUCT
		Cmd : ConvHandOffCmdTyp;
		Par : ConvHandOffParTyp;
		Sts : ConvHandOffStsTyp;
	END_STRUCT;
	ConvHandOffCmdTyp : 	STRUCT
		SetupZone : BOOL;
		DeleteZone : BOOL;
		Offload : BOOL;
		Reset : BOOL;
	END_STRUCT;
	ConvHandOffParTyp : 	STRUCT
		ShuttleID : USINT;
		ZonePars : ZoneParsTyp;
	END_STRUCT;
	ConvHandOffStsTyp : 	STRUCT
		ZoneSts : McAcp6DZoneStatusType;
		Ready : BOOL;
	END_STRUCT;
	ConvHandOffStateEnum :
		(
		HAND_IDLE,
		HAND_SETUP_ZONE,
		HAND_ACTIVATE_ZONE,
		HAND_GET_ZONE_STATUS,
		HAND_WAIT,
		HAND_MOVE_SHUTTLE_ENTRANCE,
		HAND_UNLOAD_SHUTTLE,
		HAND_DEACTIVATE_ZONE,
		HAND_DELETE_ZONE,
		HAND_ERROR
		);
	ZoneParsTyp : 	STRUCT
		ZoneID : USINT;
		ZoneMode : USINT;
		UnloadingMode : USINT;
		ZoneCenterX : REAL;
		ZoneCenterY : REAL;
		ZoneLength : REAL;
		ZoneWidth : REAL;
		MaxShuttleX : REAL;
		MaxShuttleY : REAL;
		Velocity : REAL;
		Accel : REAL;
	END_STRUCT;
	HandOffFbsTyp : 	STRUCT
		ZoneCreateFb : MC_BR_ZoneCreate_Acp6D;
		ZoneDeactivateFb : MC_BR_ZoneDeactivate_Acp6D;
		ZoneDeleteFb : MC_BR_ZoneDelete_Acp6D;
		ZoneActivateFb : MC_BR_ZoneActivate_Acp6D;
		ZoneGetStsFb : MC_BR_ZoneGetStatus_Acp6D;
		ZoneUnloadFb : MC_BR_ZoneUnload_Acp6D;
		MoveInPlane : MC_BR_MoveInPlane_Acp6D;
	END_STRUCT;
END_TYPE
```

#### Variables.var
```iecst
VAR
	state : ConvHandOffStateEnum;
	interlinkIf : ConvHandOffIfTyp;
	fbs : HandOffFbsTyp;
END_VAR
```

#### Cyclic.st
```iecst
(*
	Program to control interfacing with a conveyor to unload a shuttle

	Steps
		Setup Unload Zone
		Get UnloadZone Status to get entry point
		Command shuttle to entry point
		Issue ZoneUnload
*)

PROGRAM _CYCLIC
	CASE state OF
		HAND_IDLE:
			IF interlinkIf.Cmd.SetupZone THEN
				fbs.ZoneCreateFb.Controller := ADR(gMcAcp6DController);
				fbs.ZoneCreateFb.ZoneID := interlinkIf.Par.ZonePars.ZoneID;
				fbs.ZoneCreateFb.ZoneMode := interlinkIf.Par.ZonePars.ZoneMode;
				fbs.ZoneCreateFb.UnloadingMode := interlinkIf.Par.ZonePars.UnloadingMode;
				fbs.ZoneCreateFb.ZoneCenterX := interlinkIf.Par.ZonePars.ZoneCenterX;
				fbs.ZoneCreateFb.ZoneCenterY := interlinkIf.Par.ZonePars.ZoneCenterY;
				fbs.ZoneCreateFb.ZoneLength := interlinkIf.Par.ZonePars.ZoneLength;
				fbs.ZoneCreateFb.ZoneWidth := interlinkIf.Par.ZonePars.ZoneWidth;
				fbs.ZoneCreateFb.MaxShuttleSizeX := interlinkIf.Par.ZonePars.MaxShuttleX;
				fbs.ZoneCreateFb.MaxShuttleSizeY := interlinkIf.Par.ZonePars.MaxShuttleY;
				fbs.ZoneCreateFb.Velocity := interlinkIf.Par.ZonePars.Velocity;
				fbs.ZoneCreateFb.Acceleration := interlinkIf.Par.ZonePars.Accel;
				fbs.ZoneCreateFb.Execute := TRUE;

				state := HAND_SETUP_ZONE;
			END_IF

		HAND_SETUP_ZONE:
			IF fbs.ZoneCreateFb.Error THEN
				state := HAND_ERROR;
			ELSIF fbs.ZoneCreateFb.Done THEN
				fbs.ZoneCreateFb.Execute := FALSE;

				fbs.ZoneActivateFb.ZoneID := interlinkIf.Par.ZonePars.ZoneID;
				fbs.ZoneActivateFb.Controller := ADR(gMcAcp6DController);
				fbs.ZoneActivateFb.Execute := TRUE;

				state := HAND_ACTIVATE_ZONE;
			END_IF
		HAND_ACTIVATE_ZONE:
			IF fbs.ZoneActivateFb.Error THEN
				state := HAND_ERROR;
			ELSIF fbs.ZoneActivateFb.Done THEN
				fbs.ZoneActivateFb.Execute := FALSE;

				fbs.ZoneGetStsFb.Controller := ADR(gMcAcp6DController);
				fbs.ZoneGetStsFb.ZoneID := interlinkIf.Par.ZonePars.ZoneID;
				fbs.ZoneGetStsFb.Execute := TRUE;

				state := HAND_GET_ZONE_STATUS;
			END_IF
		HAND_GET_ZONE_STATUS:
			IF fbs.ZoneGetStsFb.Error THEN
				state := HAND_ERROR;
			ELSIF fbs.ZoneGetStsFb.Done THEN
				fbs.ZoneGetStsFb.Execute := FALSE;
				interlinkIf.Sts.ZoneSts := fbs.ZoneGetStsFb.ZoneStatus;
				interlinkIf.Sts.Ready := TRUE;
				interlinkIf.Cmd.SetupZone := FALSE;

				state := HAND_WAIT;
			END_IF
		HAND_WAIT:
			IF interlinkIf.Cmd.Offload THEN
				fbs.MoveInPlane.Controller := ADR(gMcAcp6DController);
				fbs.MoveInPlane.ShuttleID := interlinkIf.Par.ShuttleID+1;
				fbs.MoveInPlane.PositionX := interlinkIf.Sts.ZoneSts.ZoneX;
				fbs.MoveInPlane.PositionY := interlinkIf.Sts.ZoneSts.ZoneY;
				fbs.MoveInPlane.Velocity := interlinkIf.Par.ZonePars.Velocity;
				fbs.MoveInPlane.Acceleration := interlinkIf.Par.ZonePars.Accel;
				fbs.MoveInPlane.Execute := TRUE;

				state := HAND_MOVE_SHUTTLE_ENTRANCE;
			ELSIF interlinkIf.Cmd.DeleteZone THEN
				fbs.ZoneDeactivateFb.Controller := ADR(gMcAcp6DController);
				fbs.ZoneDeactivateFb.ZoneID := interlinkIf.Par.ZonePars.ZoneID;
				fbs.ZoneDeactivateFb.Execute := TRUE;

				state := HAND_DEACTIVATE_ZONE;
			END_IF

		HAND_MOVE_SHUTTLE_ENTRANCE:
			IF fbs.MoveInPlane.Error THEN
				state := HAND_ERROR;
			ELSIF fbs.MoveInPlane.Done THEN
				fbs.MoveInPlane.Execute := FALSE;

				fbs.ZoneUnloadFb.Controller := ADR(gMcAcp6DController);
				fbs.ZoneUnloadFb.ShuttleID := interlinkIf.Par.ShuttleID+1;
				fbs.ZoneUnloadFb.ZoneID := interlinkIf.Par.ZonePars.ZoneID;
				fbs.ZoneUnloadFb.Execute := TRUE;

				state := HAND_UNLOAD_SHUTTLE;
			END_IF

		HAND_UNLOAD_SHUTTLE:
			IF fbs.ZoneUnloadFb.Error THEN
				state := HAND_ERROR;
			ELSIF fbs.ZoneUnloadFb.Done THEN
				fbs.ZoneUnloadFb.Execute := FALSE;

				interlinkIf.Cmd.Offload := FALSE;
				state := HAND_WAIT;
			END_IF
		HAND_DEACTIVATE_ZONE:
			IF fbs.ZoneDeactivateFb.Error THEN
				state := HAND_ERROR;
			ELSIF fbs.ZoneDeactivateFb.Done THEN
				fbs.ZoneDeactivateFb.Execute := FALSE;

				fbs.ZoneDeleteFb.Controller := ADR(gMcAcp6DController);
				fbs.ZoneDeleteFb.ZoneID := interlinkIf.Par.ZonePars.ZoneID;
				fbs.ZoneDeleteFb.Execute := TRUE;

				state := HAND_DELETE_ZONE;
			END_IF
		HAND_DELETE_ZONE:
			IF fbs.ZoneDeleteFb.Error THEN
				state := HAND_ERROR;
			ELSIF fbs.ZoneDeleteFb.Done THEN
				fbs.ZoneDeleteFb.Execute := FALSE;
				interlinkIf.Sts.Ready := FALSE;

				state := HAND_IDLE;
			END_IF
		HAND_ERROR:
			IF interlinkIf.Cmd.Reset THEN
				fbs.ZoneActivateFb.Execute := FALSE;
				fbs.ZoneGetStsFb.Execute := FALSE;
				fbs.ZoneCreateFb.Execute := FALSE;
				fbs.MoveInPlane.Execute := FALSE;
				fbs.ZoneUnloadFb.Execute := FALSE;
				fbs.ZoneDeleteFb.Execute := FALSE;
				fbs.ZoneDeactivateFb.Execute := FALSE;

				interlinkIf.Cmd.Offload := FALSE;
				interlinkIf.Cmd.Reset := FALSE;
				interlinkIf.Cmd.SetupZone := FALSE;

				IF interlinkIf.Sts.Ready THEN
					state := HAND_WAIT;
				ELSE
					state := HAND_IDLE;
				END_IF

			END_IF
	END_CASE;

	fbs.ZoneActivateFb();
	fbs.ZoneDeleteFb();
	fbs.ZoneDeactivateFb();
	fbs.ZoneGetStsFb();
	fbs.ZoneCreateFb();
	fbs.MoveInPlane();
	fbs.ZoneUnloadFb();
END_PROGRAM
```

#### Init.st
```iecst
PROGRAM _INIT

	interlinkIf.Par.ZonePars.ZoneCenterX := 0.0;
	interlinkIf.Par.ZonePars.ZoneCenterY := 0.12;
	interlinkIf.Par.ZonePars.ZoneWidth := 0.12;
	interlinkIf.Par.ZonePars.ZoneLength := 0.12;
	interlinkIf.Par.ZonePars.ZoneID := 1;
	interlinkIf.Par.ZonePars.Velocity := 0.5;
	interlinkIf.Par.ZonePars.Accel := 10;
	interlinkIf.Par.ZonePars.MaxShuttleX := 0.12;
	interlinkIf.Par.ZonePars.MaxShuttleY := 0.12;
	interlinkIf.Par.ZonePars.ZoneMode := 0;

END_PROGRAM
```

### Program Logical/Source/Demos/GenMoveDemo (IEC)

#### Types.typ - Local data types
```iecst
TYPE
	GenMoveDemoIf : 	STRUCT
		Cmds : GenMoveDemoIfCmdTyp;
		Sts : GenMoveIfStsTyp;
	END_STRUCT;
	GenMoveDemoIfCmdTyp : 	STRUCT
		RunDemo : BOOL;
		Reset : BOOL;
	END_STRUCT;
	GenMoveIfParTyp : 	STRUCT
	END_STRUCT;
	GenMoveIfStsTyp : 	STRUCT
		Running : BOOL;
	END_STRUCT;
	GenMoveIfStateEnum :
		(
		GEN_IDLE,
		GEN_INIT,
		GEN_LAPS,
		GEN_ORBIT,
		GEN_SQUARE,
		GEN_COUPLED_LAP,
		GEN_CIRCLE,
		GEN_6DOF,
		GEN_ERROR
		);
	GenMoveFbsTyp : 	STRUCT
	END_STRUCT;
END_TYPE
```

#### LocalFunctions.fun
```iecst
{REDUND_ERROR} FUNCTION_BLOCK genLapsFb (*Runs a 2 shuttle lap demo on a 1x2 6d layout*) (*$GROUP=User,$CAT=User,$GROUPICON=User.png,$CATICON=User.png*)
	VAR_INPUT
		Execute : {REDUND_UNREPLICABLE} BOOL;
		Controller : REFERENCE TO McAcp6DControllerType;
		Velocity : REAL;
		Accel : REAL;
		NumLaps : USINT;
	END_VAR
	VAR_OUTPUT
		Active : {REDUND_UNREPLICABLE} BOOL;
		Done : {REDUND_UNREPLICABLE} BOOL;
		Error : {REDUND_UNREPLICABLE} BOOL;
	END_VAR
	VAR
		internal : {REDUND_UNREPLICABLE} BOOL;
	END_VAR
END_FUNCTION_BLOCK
```

#### LocalFunctionsTypes.typ - Local data types
```iecst
(*Laps Internal Type*)

TYPE
	GenLapsDemoInternalTyp : 	STRUCT
		state : USINT;
		lapCounter : USINT;
		Fbs : USINT;
	END_STRUCT;
	GenLapsDemoFbsTyp : 	STRUCT
		AsyncMoveFb : MC_BR_MoveInPlaneAsync_Acp6D;
		MovePlaneFb : MC_BR_MoveInPlane_Acp6D;
		MoveArcFb : MC_BR_MoveArcAngle_Acp6D;
		BufferCtrlFb : MC_BR_BufferCtrl_Acp6D;
	END_STRUCT;
	GenLapsStateEnum :
		(
		LAPS_OFF, (*Off state*)
		LAPS_INIT, (*Init state*)
		LAPS_ASYNC_WAIT, (*Waiting for Aysync Move to complete*)
		LAPS_BLOCK_BUFFER, (*Waiting for Block Cmd*)
		LAPS_MOVE_OVER,
		LAPS_MOVE_ARC,
		LAPS_MOVE_OVER2,
		LAPS_MOVE_ARC2,
		LAPS_RELEASE_BUFFER,
		LAPS_DONE,
		LAPS_ERROR
		);
END_TYPE
```

#### genLapsFb.st
```iecst
(* Runs a 2 shuttle lap demo on a 1x2 6d layout *)
FUNCTION_BLOCK genLapsFb
END_FUNCTION_BLOCK
```

- gAssembly_1.wsp (not shown)

- Visualisation Logical/mappView (not shown)

Listed in the project but not available here: Logical/Global.typ, Logical/Global.var, Logical/Source/ShuttleCtrl/ShCtrlGlobalVars.var, Logical/Source/ShuttleCtrl/ShCtrlGlobalTypes.typ, Logical/Source/ProcessStations/ProCGlobalTypes.typ, Logical/Source/ProcessStations/ProcGlobalVars.var, Logical/Source/Demos/GenMoveDemo/Cyclic.st, Logical/Source/Demos/GenMoveDemo/Init.st, Logical/Source/Demos/GenMoveDemo/Exit.st, Logical/Source/Demos/GenMoveDemo/Variables.var, Logical/Source/Demos/GenMoveDemo/LocalFunctionVars.var
